// TIA Portal V19 export
FUNCTION "MANUAL INTERLOCK" : Void   // FC8, LAD
{ S7_Optimized_Access := 'TRUE' }
// stored: SetENOAutomatically false
BEGIN

REGION Network 1: ERROR BIT
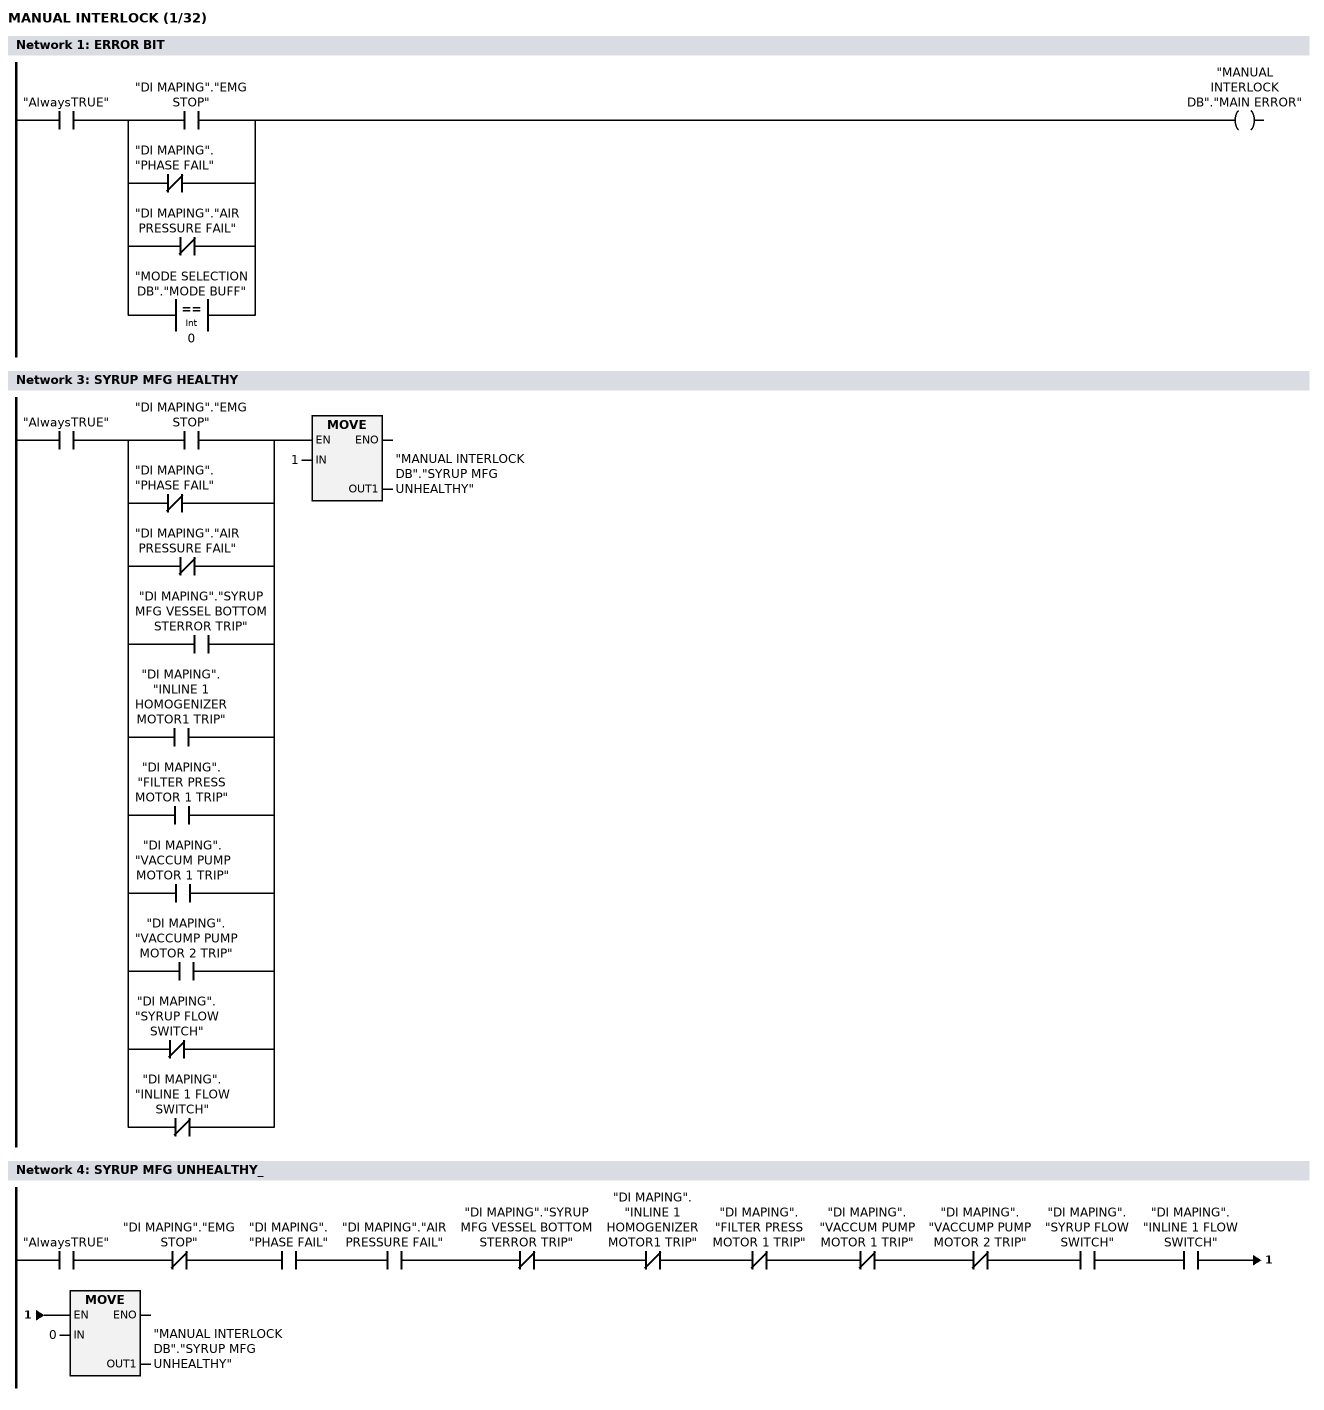
   RUNG wire#powerrail
      Contact( "AlwaysTRUE" )
      wire#w1
      Contact( "DI MAPING"."EMG STOP" )
      wire#w2
      Coil( "MANUAL INTERLOCK DB"."MAIN ERROR" )
   END_RUNG
   RUNG wire#w1
      I_Contact( "DI MAPING"."PHASE FAIL" )
   END_RUNG wire#w2
   RUNG wire#w1
      I_Contact( "DI MAPING"."AIR PRESSURE FAIL" )
   END_RUNG wire#w2
   RUNG wire#w1
      { S7_Templates := "SrcType := Int" } EQ_Contact(in1 := "MODE SELECTION DB"."MODE BUFF", in2 := 0)
   END_RUNG wire#w2
   // the same network as SCL:
   "MANUAL INTERLOCK DB"."MAIN ERROR" := "AlwaysTRUE" AND ("DI MAPING"."EMG STOP" OR NOT "DI MAPING"."PHASE FAIL" OR NOT "DI MAPING"."AIR PRESSURE FAIL" OR ("MODE SELECTION DB"."MODE BUFF" = 0));
END_REGION

REGION Network 3: SYRUP MFG HEALTHY
   RUNG wire#powerrail
      Contact( "AlwaysTRUE" )
      wire#w1
      Contact( "DI MAPING"."EMG STOP" )
      wire#w2
      Move(in := 1, out1 => "MANUAL INTERLOCK DB"."SYRUP MFG UNHEALTHY")
   END_RUNG
   RUNG wire#w1
      I_Contact( "DI MAPING"."PHASE FAIL" )
   END_RUNG wire#w2
   RUNG wire#w1
      I_Contact( "DI MAPING"."AIR PRESSURE FAIL" )
   END_RUNG wire#w2
   RUNG wire#w1
      Contact( "DI MAPING"."SYRUP MFG VESSEL BOTTOM STERROR TRIP" )
   END_RUNG wire#w2
   RUNG wire#w1
      Contact( "DI MAPING"."INLINE 1 HOMOGENIZER MOTOR1 TRIP" )
   END_RUNG wire#w2
   RUNG wire#w1
      Contact( "DI MAPING"."FILTER PRESS MOTOR 1 TRIP" )
   END_RUNG wire#w2
   RUNG wire#w1
      Contact( "DI MAPING"."VACCUM PUMP MOTOR 1 TRIP" )
   END_RUNG wire#w2
   RUNG wire#w1
      Contact( "DI MAPING"."VACCUMP PUMP MOTOR 2 TRIP" )
   END_RUNG wire#w2
   RUNG wire#w1
      I_Contact( "DI MAPING"."SYRUP FLOW SWITCH" )
   END_RUNG wire#w2
   RUNG wire#w1
      I_Contact( "DI MAPING"."INLINE 1 FLOW SWITCH" )
   END_RUNG wire#w2
   // the same network as SCL:
   IF "AlwaysTRUE" AND ("DI MAPING"."EMG STOP" OR NOT "DI MAPING"."PHASE FAIL" OR NOT "DI MAPING"."AIR PRESSURE FAIL" OR "DI MAPING"."SYRUP MFG VESSEL BOTTOM STERROR TRIP" OR "DI MAPING"."INLINE 1 HOMOGENIZER MOTOR1 TRIP" OR "DI MAPING"."FILTER PRESS MOTOR 1 TRIP" OR "DI MAPING"."VACCUM PUMP MOTOR 1 TRIP" OR "DI MAPING"."VACCUMP PUMP MOTOR 2 TRIP" OR NOT "DI MAPING"."SYRUP FLOW SWITCH" OR NOT "DI MAPING"."INLINE 1 FLOW SWITCH") THEN
       "MANUAL INTERLOCK DB"."SYRUP MFG UNHEALTHY" := 1;
   END_IF;
END_REGION

REGION Network 4: SYRUP MFG UNHEALTHY_
   RUNG wire#powerrail
      Contact( "AlwaysTRUE" )
      I_Contact( "DI MAPING"."EMG STOP" )
      Contact( "DI MAPING"."PHASE FAIL" )
      Contact( "DI MAPING"."AIR PRESSURE FAIL" )
      I_Contact( "DI MAPING"."SYRUP MFG VESSEL BOTTOM STERROR TRIP" )
      I_Contact( "DI MAPING"."INLINE 1 HOMOGENIZER MOTOR1 TRIP" )
      I_Contact( "DI MAPING"."FILTER PRESS MOTOR 1 TRIP" )
      I_Contact( "DI MAPING"."VACCUM PUMP MOTOR 1 TRIP" )
      I_Contact( "DI MAPING"."VACCUMP PUMP MOTOR 2 TRIP" )
      Contact( "DI MAPING"."SYRUP FLOW SWITCH" )
      Contact( "DI MAPING"."INLINE 1 FLOW SWITCH" )
      Move(in := 0, out1 => "MANUAL INTERLOCK DB"."SYRUP MFG UNHEALTHY")
   END_RUNG
   // the same network as SCL:
   IF "AlwaysTRUE" AND NOT "DI MAPING"."EMG STOP" AND "DI MAPING"."PHASE FAIL" AND "DI MAPING"."AIR PRESSURE FAIL" AND NOT "DI MAPING"."SYRUP MFG VESSEL BOTTOM STERROR TRIP" AND NOT "DI MAPING"."INLINE 1 HOMOGENIZER MOTOR1 TRIP" AND NOT "DI MAPING"."FILTER PRESS MOTOR 1 TRIP" AND NOT "DI MAPING"."VACCUM PUMP MOTOR 1 TRIP" AND NOT "DI MAPING"."VACCUMP PUMP MOTOR 2 TRIP" AND "DI MAPING"."SYRUP FLOW SWITCH" AND "DI MAPING"."INLINE 1 FLOW SWITCH" THEN
       "MANUAL INTERLOCK DB"."SYRUP MFG UNHEALTHY" := 0;
   END_IF;
END_REGION

REGION Network 5: PREMIXING HEALTHY
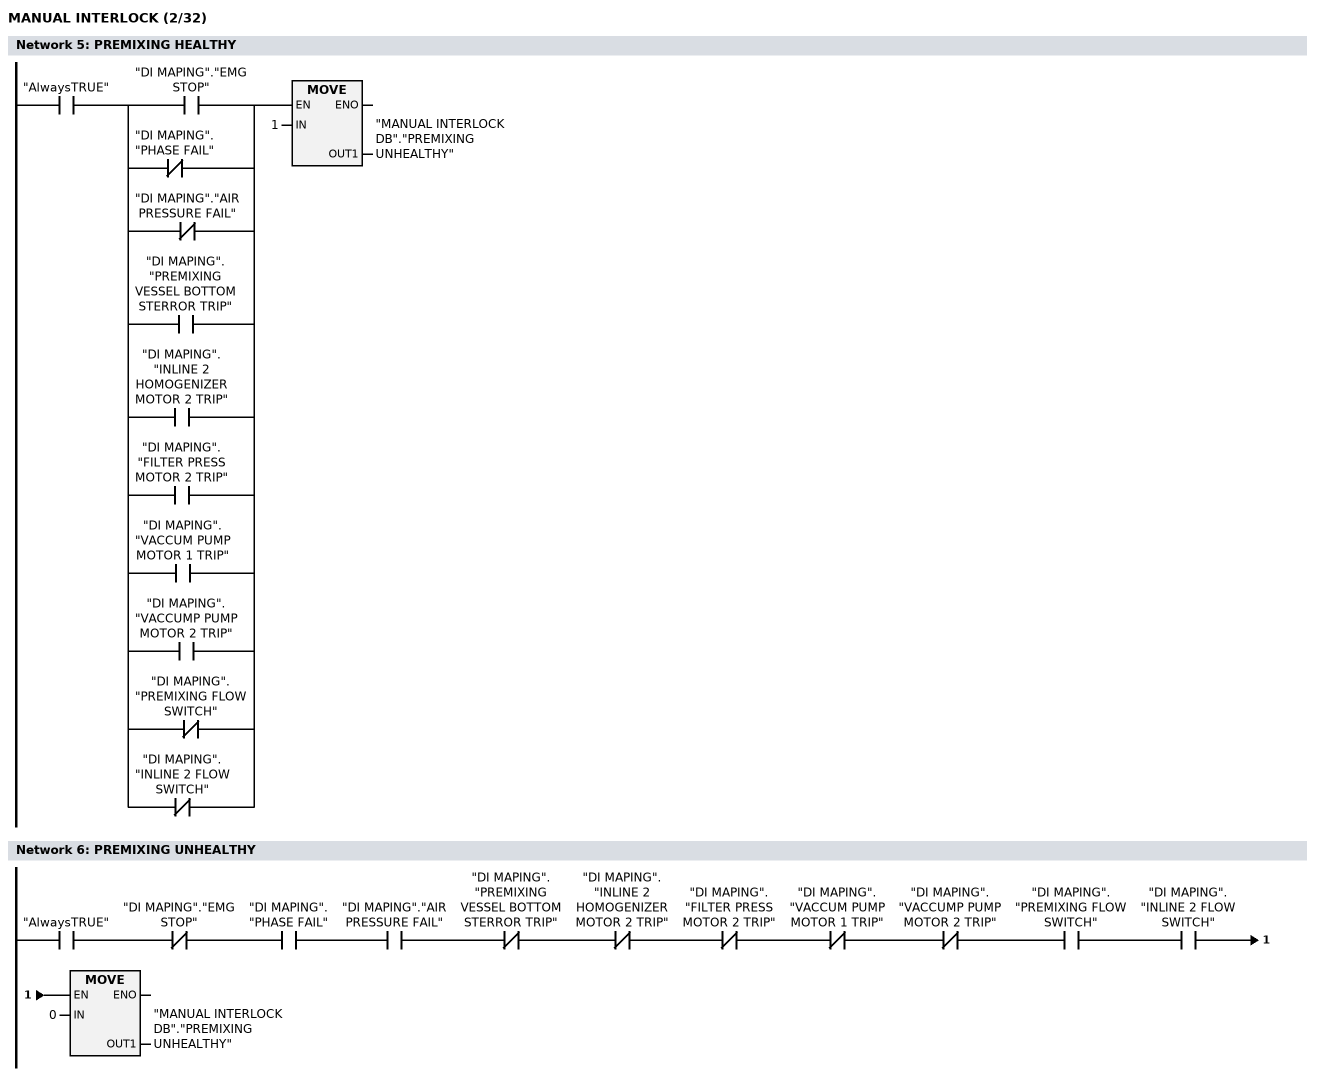
   RUNG wire#powerrail
      Contact( "AlwaysTRUE" )
      wire#w1
      Contact( "DI MAPING"."EMG STOP" )
      wire#w2
      Move(in := 1, out1 => "MANUAL INTERLOCK DB"."PREMIXING UNHEALTHY")
   END_RUNG
   RUNG wire#w1
      I_Contact( "DI MAPING"."PHASE FAIL" )
   END_RUNG wire#w2
   RUNG wire#w1
      I_Contact( "DI MAPING"."AIR PRESSURE FAIL" )
   END_RUNG wire#w2
   RUNG wire#w1
      Contact( "DI MAPING"."PREMIXING VESSEL BOTTOM STERROR TRIP" )
   END_RUNG wire#w2
   RUNG wire#w1
      Contact( "DI MAPING"."INLINE 2 HOMOGENIZER MOTOR 2 TRIP" )
   END_RUNG wire#w2
   RUNG wire#w1
      Contact( "DI MAPING"."FILTER PRESS MOTOR 2 TRIP" )
   END_RUNG wire#w2
   RUNG wire#w1
      Contact( "DI MAPING"."VACCUM PUMP MOTOR 1 TRIP" )
   END_RUNG wire#w2
   RUNG wire#w1
      Contact( "DI MAPING"."VACCUMP PUMP MOTOR 2 TRIP" )
   END_RUNG wire#w2
   RUNG wire#w1
      I_Contact( "DI MAPING"."PREMIXING FLOW SWITCH" )
   END_RUNG wire#w2
   RUNG wire#w1
      I_Contact( "DI MAPING"."INLINE 2 FLOW SWITCH" )
   END_RUNG wire#w2
   // the same network as SCL:
   IF "AlwaysTRUE" AND ("DI MAPING"."EMG STOP" OR NOT "DI MAPING"."PHASE FAIL" OR NOT "DI MAPING"."AIR PRESSURE FAIL" OR "DI MAPING"."PREMIXING VESSEL BOTTOM STERROR TRIP" OR "DI MAPING"."INLINE 2 HOMOGENIZER MOTOR 2 TRIP" OR "DI MAPING"."FILTER PRESS MOTOR 2 TRIP" OR "DI MAPING"."VACCUM PUMP MOTOR 1 TRIP" OR "DI MAPING"."VACCUMP PUMP MOTOR 2 TRIP" OR NOT "DI MAPING"."PREMIXING FLOW SWITCH" OR NOT "DI MAPING"."INLINE 2 FLOW SWITCH") THEN
       "MANUAL INTERLOCK DB"."PREMIXING UNHEALTHY" := 1;
   END_IF;
END_REGION

REGION Network 6: PREMIXING UNHEALTHY
   RUNG wire#powerrail
      Contact( "AlwaysTRUE" )
      I_Contact( "DI MAPING"."EMG STOP" )
      Contact( "DI MAPING"."PHASE FAIL" )
      Contact( "DI MAPING"."AIR PRESSURE FAIL" )
      I_Contact( "DI MAPING"."PREMIXING VESSEL BOTTOM STERROR TRIP" )
      I_Contact( "DI MAPING"."INLINE 2 HOMOGENIZER MOTOR 2 TRIP" )
      I_Contact( "DI MAPING"."FILTER PRESS MOTOR 2 TRIP" )
      I_Contact( "DI MAPING"."VACCUM PUMP MOTOR 1 TRIP" )
      I_Contact( "DI MAPING"."VACCUMP PUMP MOTOR 2 TRIP" )
      Contact( "DI MAPING"."PREMIXING FLOW SWITCH" )
      Contact( "DI MAPING"."INLINE 2 FLOW SWITCH" )
      Move(in := 0, out1 => "MANUAL INTERLOCK DB"."PREMIXING UNHEALTHY")
   END_RUNG
   // the same network as SCL:
   IF "AlwaysTRUE" AND NOT "DI MAPING"."EMG STOP" AND "DI MAPING"."PHASE FAIL" AND "DI MAPING"."AIR PRESSURE FAIL" AND NOT "DI MAPING"."PREMIXING VESSEL BOTTOM STERROR TRIP" AND NOT "DI MAPING"."INLINE 2 HOMOGENIZER MOTOR 2 TRIP" AND NOT "DI MAPING"."FILTER PRESS MOTOR 2 TRIP" AND NOT "DI MAPING"."VACCUM PUMP MOTOR 1 TRIP" AND NOT "DI MAPING"."VACCUMP PUMP MOTOR 2 TRIP" AND "DI MAPING"."PREMIXING FLOW SWITCH" AND "DI MAPING"."INLINE 2 FLOW SWITCH" THEN
       "MANUAL INTERLOCK DB"."PREMIXING UNHEALTHY" := 0;
   END_IF;
END_REGION

REGION Network 7: SUGAR HEALTHY
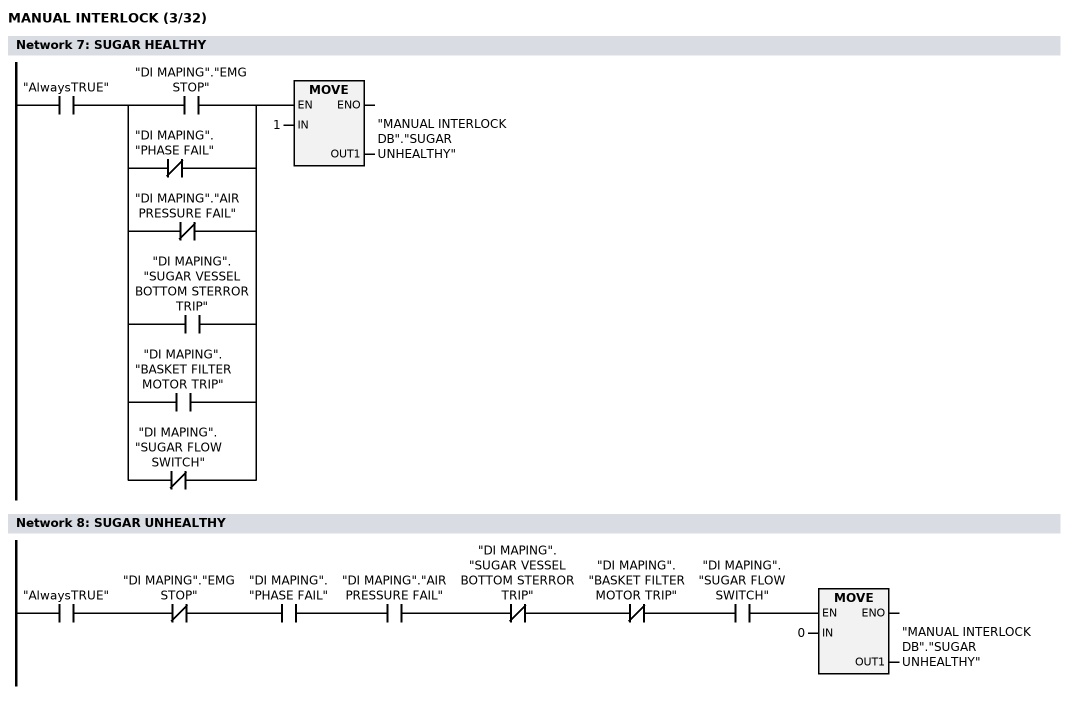
   RUNG wire#powerrail
      Contact( "AlwaysTRUE" )
      wire#w1
      Contact( "DI MAPING"."EMG STOP" )
      wire#w2
      Move(in := 1, out1 => "MANUAL INTERLOCK DB"."SUGAR UNHEALTHY")
   END_RUNG
   RUNG wire#w1
      I_Contact( "DI MAPING"."PHASE FAIL" )
   END_RUNG wire#w2
   RUNG wire#w1
      I_Contact( "DI MAPING"."AIR PRESSURE FAIL" )
   END_RUNG wire#w2
   RUNG wire#w1
      Contact( "DI MAPING"."SUGAR VESSEL BOTTOM STERROR TRIP" )
   END_RUNG wire#w2
   RUNG wire#w1
      Contact( "DI MAPING"."BASKET FILTER MOTOR TRIP" )
   END_RUNG wire#w2
   RUNG wire#w1
      I_Contact( "DI MAPING"."SUGAR FLOW SWITCH" )
   END_RUNG wire#w2
   // the same network as SCL:
   IF "AlwaysTRUE" AND ("DI MAPING"."EMG STOP" OR NOT "DI MAPING"."PHASE FAIL" OR NOT "DI MAPING"."AIR PRESSURE FAIL" OR "DI MAPING"."SUGAR VESSEL BOTTOM STERROR TRIP" OR "DI MAPING"."BASKET FILTER MOTOR TRIP" OR NOT "DI MAPING"."SUGAR FLOW SWITCH") THEN
       "MANUAL INTERLOCK DB"."SUGAR UNHEALTHY" := 1;
   END_IF;
END_REGION

REGION Network 8: SUGAR UNHEALTHY
   RUNG wire#powerrail
      Contact( "AlwaysTRUE" )
      I_Contact( "DI MAPING"."EMG STOP" )
      Contact( "DI MAPING"."PHASE FAIL" )
      Contact( "DI MAPING"."AIR PRESSURE FAIL" )
      I_Contact( "DI MAPING"."SUGAR VESSEL BOTTOM STERROR TRIP" )
      I_Contact( "DI MAPING"."BASKET FILTER MOTOR TRIP" )
      Contact( "DI MAPING"."SUGAR FLOW SWITCH" )
      Move(in := 0, out1 => "MANUAL INTERLOCK DB"."SUGAR UNHEALTHY")
   END_RUNG
   // the same network as SCL:
   IF "AlwaysTRUE" AND NOT "DI MAPING"."EMG STOP" AND "DI MAPING"."PHASE FAIL" AND "DI MAPING"."AIR PRESSURE FAIL" AND NOT "DI MAPING"."SUGAR VESSEL BOTTOM STERROR TRIP" AND NOT "DI MAPING"."BASKET FILTER MOTOR TRIP" AND "DI MAPING"."SUGAR FLOW SWITCH" THEN
       "MANUAL INTERLOCK DB"."SUGAR UNHEALTHY" := 0;
   END_IF;
END_REGION

REGION Network 10: ------------------------------------------ CONTINUE RESET-------------------------------------
END_REGION

REGION Network 11: SYRUP MFG PROCESS ERROR FOR CONTINUE
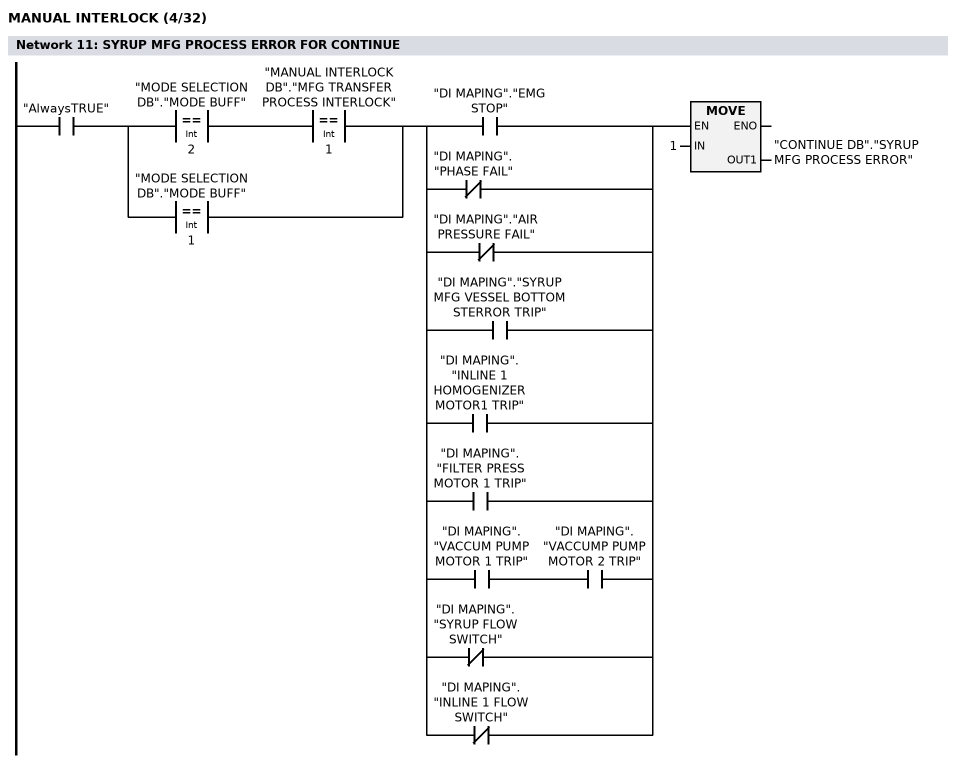
   RUNG wire#powerrail
      Contact( "AlwaysTRUE" )
      wire#w1
      { S7_Templates := "SrcType := Int" } EQ_Contact(in1 := "MODE SELECTION DB"."MODE BUFF", in2 := 2)
      { S7_Templates := "SrcType := Int" } EQ_Contact(in1 := "MANUAL INTERLOCK DB"."MFG TRANSFER PROCESS INTERLOCK", in2 := 1)
      wire#w2
      Contact( "DI MAPING"."EMG STOP" )
      wire#w3
      Move(in := 1, out1 => "CONTINUE DB"."SYRUP MFG PROCESS ERROR")
   END_RUNG
   RUNG wire#w1
      { S7_Templates := "SrcType := Int" } EQ_Contact(in1 := "MODE SELECTION DB"."MODE BUFF", in2 := 1)
   END_RUNG wire#w2
   RUNG wire#w2
      I_Contact( "DI MAPING"."PHASE FAIL" )
   END_RUNG wire#w3
   RUNG wire#w2
      I_Contact( "DI MAPING"."AIR PRESSURE FAIL" )
   END_RUNG wire#w3
   RUNG wire#w2
      Contact( "DI MAPING"."SYRUP MFG VESSEL BOTTOM STERROR TRIP" )
   END_RUNG wire#w3
   RUNG wire#w2
      Contact( "DI MAPING"."INLINE 1 HOMOGENIZER MOTOR1 TRIP" )
   END_RUNG wire#w3
   RUNG wire#w2
      Contact( "DI MAPING"."FILTER PRESS MOTOR 1 TRIP" )
   END_RUNG wire#w3
   RUNG wire#w2
      Contact( "DI MAPING"."VACCUM PUMP MOTOR 1 TRIP" )
      Contact( "DI MAPING"."VACCUMP PUMP MOTOR 2 TRIP" )
   END_RUNG wire#w3
   RUNG wire#w2
      I_Contact( "DI MAPING"."SYRUP FLOW SWITCH" )
   END_RUNG wire#w3
   RUNG wire#w2
      I_Contact( "DI MAPING"."INLINE 1 FLOW SWITCH" )
   END_RUNG wire#w3
   // the same network as SCL:
   IF "AlwaysTRUE" AND ((("MODE SELECTION DB"."MODE BUFF" = 2) AND ("MANUAL INTERLOCK DB"."MFG TRANSFER PROCESS INTERLOCK" = 1)) OR ("MODE SELECTION DB"."MODE BUFF" = 1)) AND ("DI MAPING"."EMG STOP" OR NOT "DI MAPING"."PHASE FAIL" OR NOT "DI MAPING"."AIR PRESSURE FAIL" OR "DI MAPING"."SYRUP MFG VESSEL BOTTOM STERROR TRIP" OR "DI MAPING"."INLINE 1 HOMOGENIZER MOTOR1 TRIP" OR "DI MAPING"."FILTER PRESS MOTOR 1 TRIP" OR ("DI MAPING"."VACCUM PUMP MOTOR 1 TRIP" AND "DI MAPING"."VACCUMP PUMP MOTOR 2 TRIP") OR NOT "DI MAPING"."SYRUP FLOW SWITCH" OR NOT "DI MAPING"."INLINE 1 FLOW SWITCH") THEN
       "CONTINUE DB"."SYRUP MFG PROCESS ERROR" := 1;
   END_IF;
END_REGION

REGION Network 12: PREMIXING PROCESS ERROR FOR CONTINUE
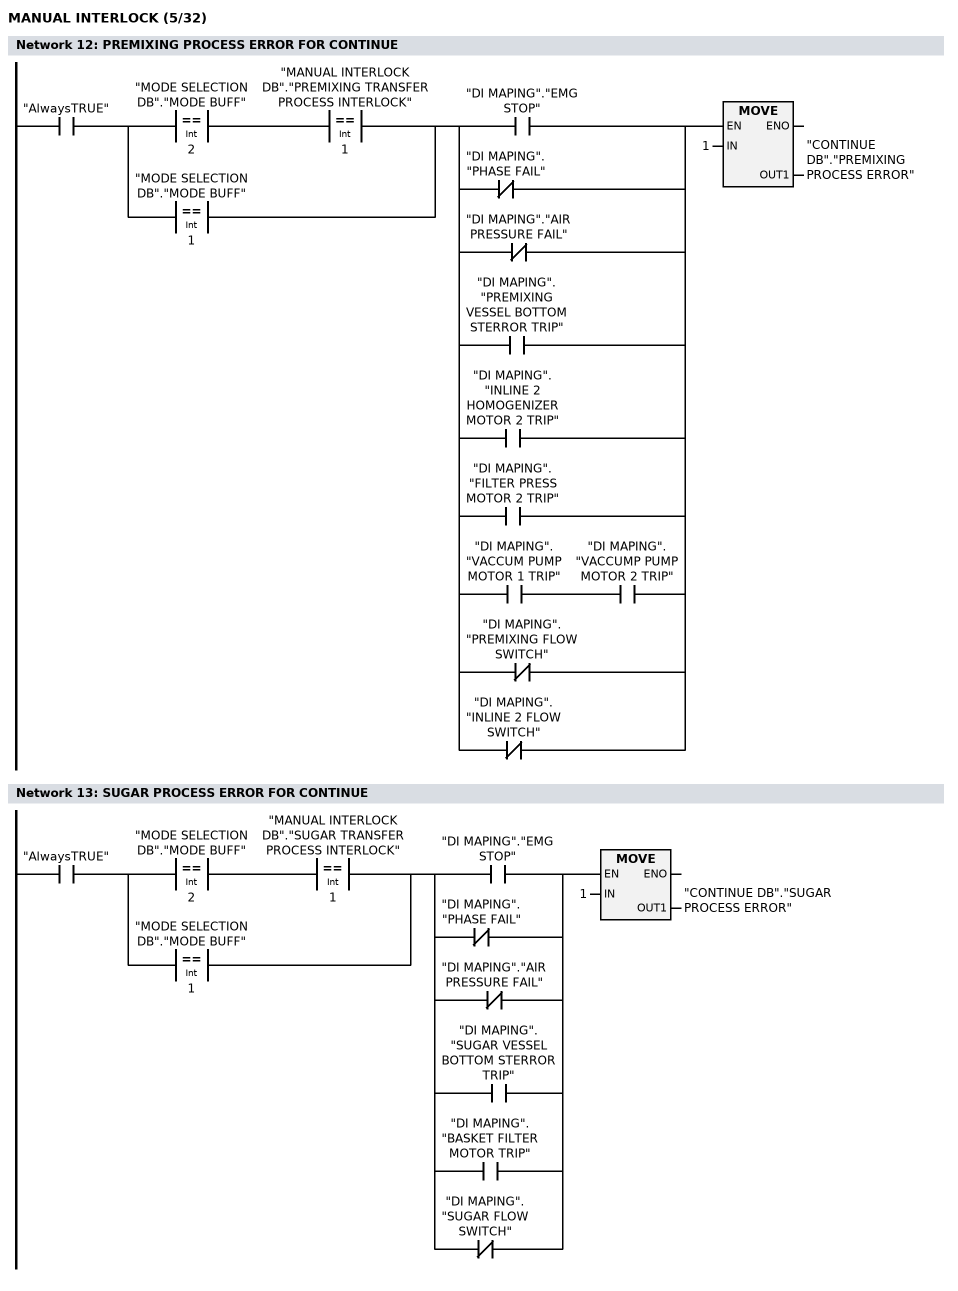
   RUNG wire#powerrail
      Contact( "AlwaysTRUE" )
      wire#w1
      { S7_Templates := "SrcType := Int" } EQ_Contact(in1 := "MODE SELECTION DB"."MODE BUFF", in2 := 2)
      { S7_Templates := "SrcType := Int" } EQ_Contact(in1 := "MANUAL INTERLOCK DB"."PREMIXING TRANSFER PROCESS INTERLOCK", in2 := 1)
      wire#w2
      Contact( "DI MAPING"."EMG STOP" )
      wire#w3
      Move(in := 1, out1 => "CONTINUE DB"."PREMIXING PROCESS ERROR")
   END_RUNG
   RUNG wire#w1
      { S7_Templates := "SrcType := Int" } EQ_Contact(in1 := "MODE SELECTION DB"."MODE BUFF", in2 := 1)
   END_RUNG wire#w2
   RUNG wire#w2
      I_Contact( "DI MAPING"."PHASE FAIL" )
   END_RUNG wire#w3
   RUNG wire#w2
      I_Contact( "DI MAPING"."AIR PRESSURE FAIL" )
   END_RUNG wire#w3
   RUNG wire#w2
      Contact( "DI MAPING"."PREMIXING VESSEL BOTTOM STERROR TRIP" )
   END_RUNG wire#w3
   RUNG wire#w2
      Contact( "DI MAPING"."INLINE 2 HOMOGENIZER MOTOR 2 TRIP" )
   END_RUNG wire#w3
   RUNG wire#w2
      Contact( "DI MAPING"."FILTER PRESS MOTOR 2 TRIP" )
   END_RUNG wire#w3
   RUNG wire#w2
      Contact( "DI MAPING"."VACCUM PUMP MOTOR 1 TRIP" )
      Contact( "DI MAPING"."VACCUMP PUMP MOTOR 2 TRIP" )
   END_RUNG wire#w3
   RUNG wire#w2
      I_Contact( "DI MAPING"."PREMIXING FLOW SWITCH" )
   END_RUNG wire#w3
   RUNG wire#w2
      I_Contact( "DI MAPING"."INLINE 2 FLOW SWITCH" )
   END_RUNG wire#w3
   // the same network as SCL:
   IF "AlwaysTRUE" AND ((("MODE SELECTION DB"."MODE BUFF" = 2) AND ("MANUAL INTERLOCK DB"."PREMIXING TRANSFER PROCESS INTERLOCK" = 1)) OR ("MODE SELECTION DB"."MODE BUFF" = 1)) AND ("DI MAPING"."EMG STOP" OR NOT "DI MAPING"."PHASE FAIL" OR NOT "DI MAPING"."AIR PRESSURE FAIL" OR "DI MAPING"."PREMIXING VESSEL BOTTOM STERROR TRIP" OR "DI MAPING"."INLINE 2 HOMOGENIZER MOTOR 2 TRIP" OR "DI MAPING"."FILTER PRESS MOTOR 2 TRIP" OR ("DI MAPING"."VACCUM PUMP MOTOR 1 TRIP" AND "DI MAPING"."VACCUMP PUMP MOTOR 2 TRIP") OR NOT "DI MAPING"."PREMIXING FLOW SWITCH" OR NOT "DI MAPING"."INLINE 2 FLOW SWITCH") THEN
       "CONTINUE DB"."PREMIXING PROCESS ERROR" := 1;
   END_IF;
END_REGION

REGION Network 13: SUGAR PROCESS ERROR FOR CONTINUE
   RUNG wire#powerrail
      Contact( "AlwaysTRUE" )
      wire#w1
      { S7_Templates := "SrcType := Int" } EQ_Contact(in1 := "MODE SELECTION DB"."MODE BUFF", in2 := 2)
      { S7_Templates := "SrcType := Int" } EQ_Contact(in1 := "MANUAL INTERLOCK DB"."SUGAR TRANSFER PROCESS INTERLOCK", in2 := 1)
      wire#w2
      Contact( "DI MAPING"."EMG STOP" )
      wire#w3
      Move(in := 1, out1 => "CONTINUE DB"."SUGAR PROCESS ERROR")
   END_RUNG
   RUNG wire#w1
      { S7_Templates := "SrcType := Int" } EQ_Contact(in1 := "MODE SELECTION DB"."MODE BUFF", in2 := 1)
   END_RUNG wire#w2
   RUNG wire#w2
      I_Contact( "DI MAPING"."PHASE FAIL" )
   END_RUNG wire#w3
   RUNG wire#w2
      I_Contact( "DI MAPING"."AIR PRESSURE FAIL" )
   END_RUNG wire#w3
   RUNG wire#w2
      Contact( "DI MAPING"."SUGAR VESSEL BOTTOM STERROR TRIP" )
   END_RUNG wire#w3
   RUNG wire#w2
      Contact( "DI MAPING"."BASKET FILTER MOTOR TRIP" )
   END_RUNG wire#w3
   RUNG wire#w2
      I_Contact( "DI MAPING"."SUGAR FLOW SWITCH" )
   END_RUNG wire#w3
   // the same network as SCL:
   IF "AlwaysTRUE" AND ((("MODE SELECTION DB"."MODE BUFF" = 2) AND ("MANUAL INTERLOCK DB"."SUGAR TRANSFER PROCESS INTERLOCK" = 1)) OR ("MODE SELECTION DB"."MODE BUFF" = 1)) AND ("DI MAPING"."EMG STOP" OR NOT "DI MAPING"."PHASE FAIL" OR NOT "DI MAPING"."AIR PRESSURE FAIL" OR "DI MAPING"."SUGAR VESSEL BOTTOM STERROR TRIP" OR "DI MAPING"."BASKET FILTER MOTOR TRIP" OR NOT "DI MAPING"."SUGAR FLOW SWITCH") THEN
       "CONTINUE DB"."SUGAR PROCESS ERROR" := 1;
   END_IF;
END_REGION

REGION Network 15: CONTINUE PROCESS-SYRUP MFG
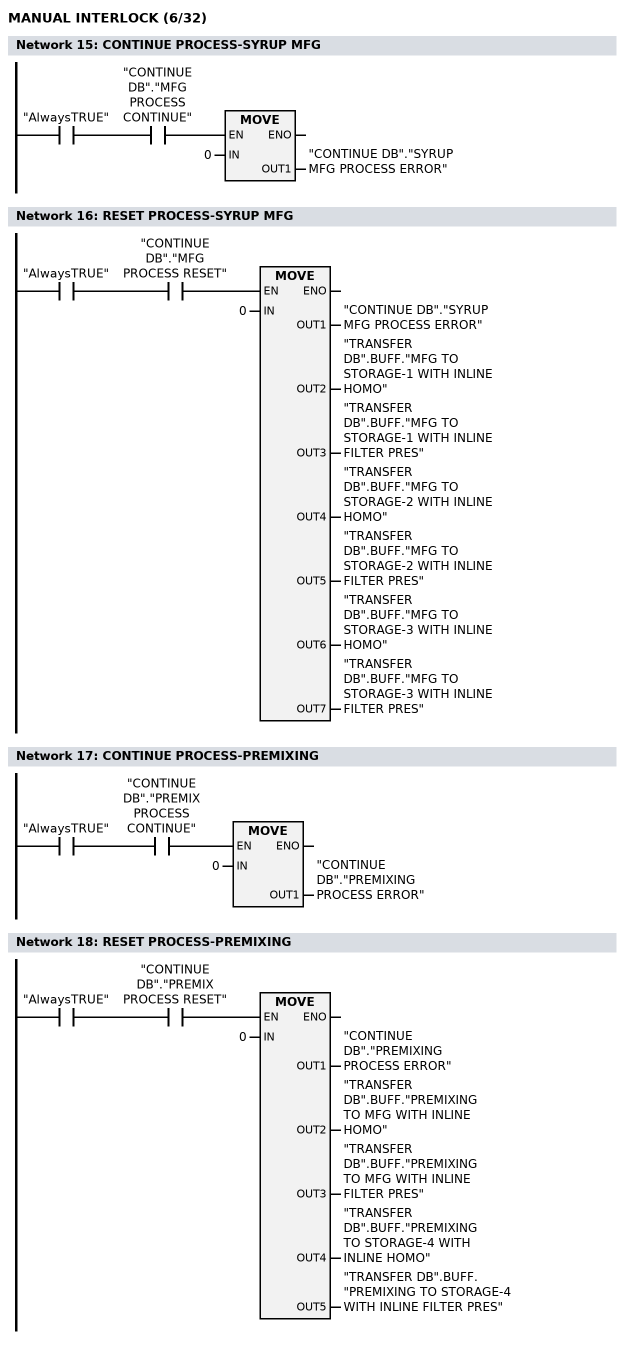
   RUNG wire#powerrail
      Contact( "AlwaysTRUE" )
      Contact( "CONTINUE DB"."MFG PROCESS CONTINUE" )
      Move(in := 0, out1 => "CONTINUE DB"."SYRUP MFG PROCESS ERROR")
   END_RUNG
   // the same network as SCL:
   IF "AlwaysTRUE" AND "CONTINUE DB"."MFG PROCESS CONTINUE" THEN
       "CONTINUE DB"."SYRUP MFG PROCESS ERROR" := 0;
   END_IF;
END_REGION

REGION Network 16: RESET PROCESS-SYRUP MFG
   RUNG wire#powerrail
      Contact( "AlwaysTRUE" )
      Contact( "CONTINUE DB"."MFG PROCESS RESET" )
      Move(in := 0, out1 => "CONTINUE DB"."SYRUP MFG PROCESS ERROR", out2 => "TRANSFER DB".BUFF."MFG TO STORAGE-1 WITH INLINE HOMO", out3 => "TRANSFER DB".BUFF."MFG TO STORAGE-1 WITH INLINE FILTER PRES", out4 => "TRANSFER DB".BUFF."MFG TO STORAGE-2 WITH INLINE HOMO", out5 => "TRANSFER DB".BUFF."MFG TO STORAGE-2 WITH INLINE FILTER PRES", out6 => "TRANSFER DB".BUFF."MFG TO STORAGE-3 WITH INLINE HOMO", out7 => "TRANSFER DB".BUFF."MFG TO STORAGE-3 WITH INLINE FILTER PRES")
   END_RUNG
   // the same network as SCL:
   IF "AlwaysTRUE" AND "CONTINUE DB"."MFG PROCESS RESET" THEN
       "CONTINUE DB"."SYRUP MFG PROCESS ERROR" := 0;
       "TRANSFER DB".BUFF."MFG TO STORAGE-1 WITH INLINE HOMO" := 0;
       "TRANSFER DB".BUFF."MFG TO STORAGE-1 WITH INLINE FILTER PRES" := 0;
       "TRANSFER DB".BUFF."MFG TO STORAGE-2 WITH INLINE HOMO" := 0;
       "TRANSFER DB".BUFF."MFG TO STORAGE-2 WITH INLINE FILTER PRES" := 0;
       "TRANSFER DB".BUFF."MFG TO STORAGE-3 WITH INLINE HOMO" := 0;
       "TRANSFER DB".BUFF."MFG TO STORAGE-3 WITH INLINE FILTER PRES" := 0;
   END_IF;
END_REGION

REGION Network 17: CONTINUE PROCESS-PREMIXING
   RUNG wire#powerrail
      Contact( "AlwaysTRUE" )
      Contact( "CONTINUE DB"."PREMIX PROCESS CONTINUE" )
      Move(in := 0, out1 => "CONTINUE DB"."PREMIXING PROCESS ERROR")
   END_RUNG
   // the same network as SCL:
   IF "AlwaysTRUE" AND "CONTINUE DB"."PREMIX PROCESS CONTINUE" THEN
       "CONTINUE DB"."PREMIXING PROCESS ERROR" := 0;
   END_IF;
END_REGION

REGION Network 18: RESET PROCESS-PREMIXING
   RUNG wire#powerrail
      Contact( "AlwaysTRUE" )
      Contact( "CONTINUE DB"."PREMIX PROCESS RESET" )
      Move(in := 0, out1 => "CONTINUE DB"."PREMIXING PROCESS ERROR", out2 => "TRANSFER DB".BUFF."PREMIXING TO MFG WITH INLINE HOMO", out3 => "TRANSFER DB".BUFF."PREMIXING TO MFG WITH INLINE FILTER PRES", out4 => "TRANSFER DB".BUFF."PREMIXING TO STORAGE-4 WITH INLINE HOMO", out5 => "TRANSFER DB".BUFF."PREMIXING TO STORAGE-4 WITH INLINE FILTER PRES")
   END_RUNG
   // the same network as SCL:
   IF "AlwaysTRUE" AND "CONTINUE DB"."PREMIX PROCESS RESET" THEN
       "CONTINUE DB"."PREMIXING PROCESS ERROR" := 0;
       "TRANSFER DB".BUFF."PREMIXING TO MFG WITH INLINE HOMO" := 0;
       "TRANSFER DB".BUFF."PREMIXING TO MFG WITH INLINE FILTER PRES" := 0;
       "TRANSFER DB".BUFF."PREMIXING TO STORAGE-4 WITH INLINE HOMO" := 0;
       "TRANSFER DB".BUFF."PREMIXING TO STORAGE-4 WITH INLINE FILTER PRES" := 0;
   END_IF;
END_REGION

REGION Network 19: CONTINUE PROCESS-SUGAR
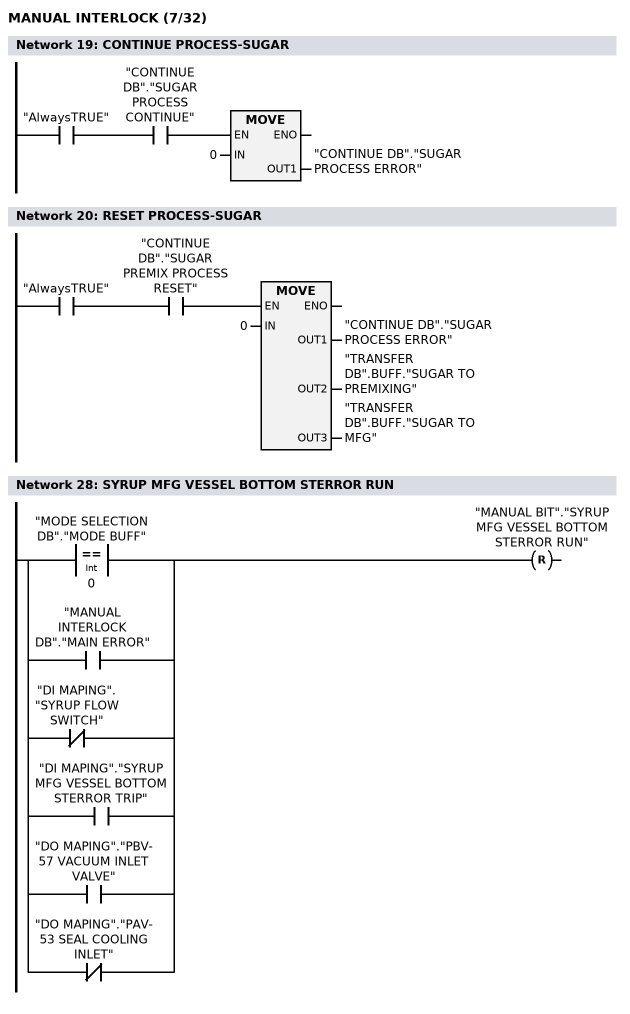
   RUNG wire#powerrail
      Contact( "AlwaysTRUE" )
      Contact( "CONTINUE DB"."SUGAR PROCESS CONTINUE" )
      Move(in := 0, out1 => "CONTINUE DB"."SUGAR PROCESS ERROR")
   END_RUNG
   // the same network as SCL:
   IF "AlwaysTRUE" AND "CONTINUE DB"."SUGAR PROCESS CONTINUE" THEN
       "CONTINUE DB"."SUGAR PROCESS ERROR" := 0;
   END_IF;
END_REGION

REGION Network 20: RESET PROCESS-SUGAR
   RUNG wire#powerrail
      Contact( "AlwaysTRUE" )
      Contact( "CONTINUE DB"."SUGAR PREMIX PROCESS RESET" )
      Move(in := 0, out1 => "CONTINUE DB"."SUGAR PROCESS ERROR", out2 => "TRANSFER DB".BUFF."SUGAR TO PREMIXING", out3 => "TRANSFER DB".BUFF."SUGAR TO MFG")
   END_RUNG
   // the same network as SCL:
   IF "AlwaysTRUE" AND "CONTINUE DB"."SUGAR PREMIX PROCESS RESET" THEN
       "CONTINUE DB"."SUGAR PROCESS ERROR" := 0;
       "TRANSFER DB".BUFF."SUGAR TO PREMIXING" := 0;
       "TRANSFER DB".BUFF."SUGAR TO MFG" := 0;
   END_IF;
END_REGION

REGION Network 22: ------------------------------TRANSFER PROCESS INTERLOCK---------------------------------------
END_REGION

REGION Network 23 (SCL): MFG TRANSFER PROCESS INTERLOCK
   IF 
       "TRANSFER DB".BUFF."MFG TO STORAGE-1 WITH INLINE HOMO" <> 0 OR
       "TRANSFER DB".BUFF."MFG TO STORAGE-1 WITH INLINE FILTER PRES" <> 0 OR
       "TRANSFER DB".BUFF."MFG TO STORAGE-2 WITH INLINE HOMO" <> 0 OR
       "TRANSFER DB".BUFF."MFG TO STORAGE-2 WITH INLINE FILTER PRES" <> 0 OR
       "TRANSFER DB".BUFF."MFG TO STORAGE-3 WITH INLINE HOMO" <> 0 OR
       "TRANSFER DB".BUFF."MFG TO STORAGE-3 WITH INLINE FILTER PRES" <> 0
   THEN
       "MANUAL INTERLOCK DB"."MFG TRANSFER PROCESS INTERLOCK" := 1;
   ELSIF "TRANSFER DB"."MFG VACCUM PUMP MOTOR-W 1 BIT"<>0
       OR "TRANSFER DB"."MFG VACCUMP PUMP MOTOR-S2 BIT"<>0
   THEN
       "MANUAL INTERLOCK DB"."MFG TRANSFER PROCESS INTERLOCK" := 2;
   ELSIF "RECIRCULATION DB".MFG.BUFF<>0
   THEN
       "MANUAL INTERLOCK DB"."MFG TRANSFER PROCESS INTERLOCK" := 3;
   ELSE
       "MANUAL INTERLOCK DB"."MFG TRANSFER PROCESS INTERLOCK" := 0;
   END_IF;
END_REGION

REGION Network 24 (SCL): PREMIXING TRANSFER PROCESS INTERLOCK
   IF
       "TRANSFER DB".BUFF."PREMIXING TO MFG WITH INLINE HOMO" <> 0 OR
       "TRANSFER DB".BUFF."PREMIXING TO MFG WITH INLINE FILTER PRES" <> 0 OR
       "TRANSFER DB".BUFF."PREMIXING TO STORAGE-4 WITH INLINE HOMO" <> 0 OR
       "TRANSFER DB".BUFF."PREMIXING TO STORAGE-4 WITH INLINE FILTER PRES" <> 0
   THEN
       "MANUAL INTERLOCK DB"."PREMIXING TRANSFER PROCESS INTERLOCK" := 1;
   ELSIF "TRANSFER DB"."PREMIXING VACCUM PUMP MOTOR-W 1 BIT"<>0 OR
       "TRANSFER DB"."PREMIXING VACCUMP PUMP MOTOR-S2 BIT"
   THEN
       "MANUAL INTERLOCK DB"."PREMIXING TRANSFER PROCESS INTERLOCK" := 2;
   ELSIF "RECIRCULATION DB".PREMIXING.BUFF<>0
   THEN
       "MANUAL INTERLOCK DB"."PREMIXING TRANSFER PROCESS INTERLOCK" := 3;
   ELSE
       "MANUAL INTERLOCK DB"."PREMIXING TRANSFER PROCESS INTERLOCK" := 0;
   END_IF;
END_REGION

REGION Network 25 (SCL): SUGAR TRANSFER PROCESS INTERLOCK
   IF "TRANSFER DB".BUFF."SUGAR TO PREMIXING" <>0 OR
       "TRANSFER DB".BUFF."SUGAR TO MFG"<>0
   THEN
       "MANUAL INTERLOCK DB"."SUGAR TRANSFER PROCESS INTERLOCK" := 1;
   ELSIF "DO MAPING"."PBV-30 VACUUM INLET VALVE" <>0
   THEN
       "MANUAL INTERLOCK DB"."SUGAR TRANSFER PROCESS INTERLOCK" := 2;
   ELSE
       "MANUAL INTERLOCK DB"."SUGAR TRANSFER PROCESS INTERLOCK" := 0;

   END_IF;
END_REGION

REGION Network 27: ------------------------------------------ MANUAL BIT RESET-------------------------------------
END_REGION

REGION Network 28: SYRUP MFG VESSEL BOTTOM STERROR RUN
   RUNG wire#powerrail
      { S7_Templates := "SrcType := Int" } EQ_Contact(in1 := "MODE SELECTION DB"."MODE BUFF", in2 := 0)
      wire#w1
      R_Coil( "MANUAL BIT"."SYRUP MFG VESSEL BOTTOM STERROR RUN" )
   END_RUNG
   RUNG wire#powerrail
      Contact( "MANUAL INTERLOCK DB"."MAIN ERROR" )
   END_RUNG wire#w1
   RUNG wire#powerrail
      I_Contact( "DI MAPING"."SYRUP FLOW SWITCH" )
   END_RUNG wire#w1
   RUNG wire#powerrail
      Contact( "DI MAPING"."SYRUP MFG VESSEL BOTTOM STERROR TRIP" )
   END_RUNG wire#w1
   RUNG wire#powerrail
      Contact( "DO MAPING"."PBV-57 VACUUM INLET VALVE" )
   END_RUNG wire#w1
   RUNG wire#powerrail
      I_Contact( "DO MAPING"."PAV-53 SEAL COOLING INLET" )
   END_RUNG wire#w1
   // the same network as SCL:
   IF ("MODE SELECTION DB"."MODE BUFF" = 0) OR "MANUAL INTERLOCK DB"."MAIN ERROR" OR NOT "DI MAPING"."SYRUP FLOW SWITCH" OR "DI MAPING"."SYRUP MFG VESSEL BOTTOM STERROR TRIP" OR "DO MAPING"."PBV-57 VACUUM INLET VALVE" OR NOT "DO MAPING"."PAV-53 SEAL COOLING INLET" THEN
       "MANUAL BIT"."SYRUP MFG VESSEL BOTTOM STERROR RUN" := FALSE;
   END_IF;
END_REGION

REGION Network 29: PREMIXING VESSEL BOTTOM STERROR RUN
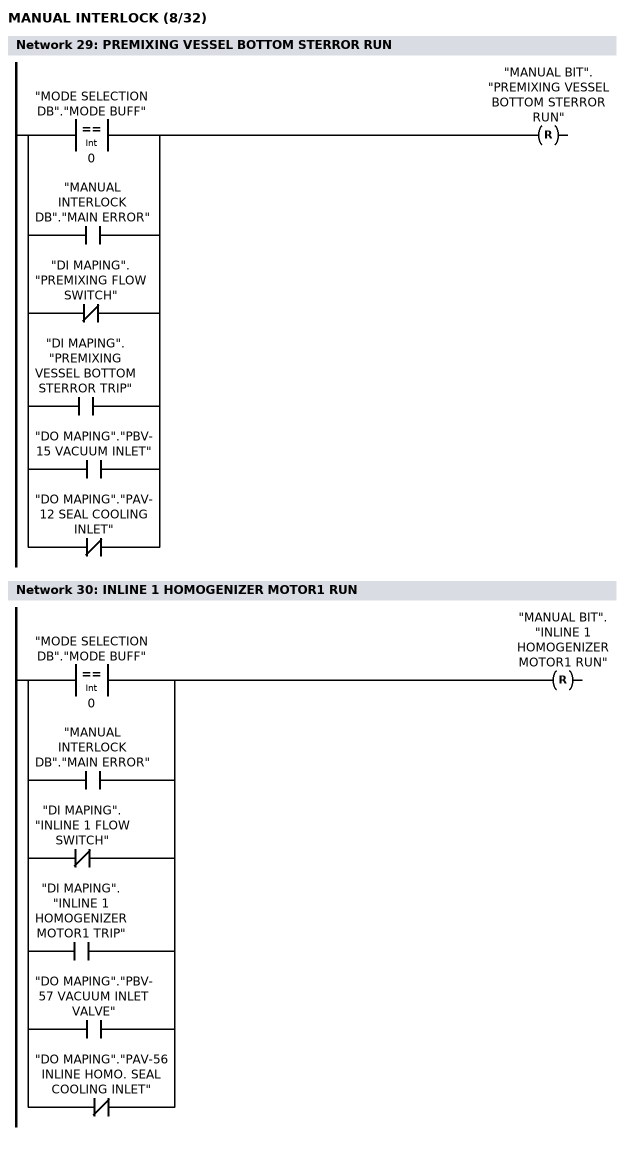
   RUNG wire#powerrail
      { S7_Templates := "SrcType := Int" } EQ_Contact(in1 := "MODE SELECTION DB"."MODE BUFF", in2 := 0)
      wire#w1
      R_Coil( "MANUAL BIT"."PREMIXING VESSEL BOTTOM STERROR RUN" )
   END_RUNG
   RUNG wire#powerrail
      Contact( "MANUAL INTERLOCK DB"."MAIN ERROR" )
   END_RUNG wire#w1
   RUNG wire#powerrail
      I_Contact( "DI MAPING"."PREMIXING FLOW SWITCH" )
   END_RUNG wire#w1
   RUNG wire#powerrail
      Contact( "DI MAPING"."PREMIXING VESSEL BOTTOM STERROR TRIP" )
   END_RUNG wire#w1
   RUNG wire#powerrail
      Contact( "DO MAPING"."PBV-15 VACUUM INLET" )
   END_RUNG wire#w1
   RUNG wire#powerrail
      I_Contact( "DO MAPING"."PAV-12 SEAL COOLING INLET" )
   END_RUNG wire#w1
   // the same network as SCL:
   IF ("MODE SELECTION DB"."MODE BUFF" = 0) OR "MANUAL INTERLOCK DB"."MAIN ERROR" OR NOT "DI MAPING"."PREMIXING FLOW SWITCH" OR "DI MAPING"."PREMIXING VESSEL BOTTOM STERROR TRIP" OR "DO MAPING"."PBV-15 VACUUM INLET" OR NOT "DO MAPING"."PAV-12 SEAL COOLING INLET" THEN
       "MANUAL BIT"."PREMIXING VESSEL BOTTOM STERROR RUN" := FALSE;
   END_IF;
END_REGION

REGION Network 30: INLINE 1 HOMOGENIZER MOTOR1 RUN
   RUNG wire#powerrail
      { S7_Templates := "SrcType := Int" } EQ_Contact(in1 := "MODE SELECTION DB"."MODE BUFF", in2 := 0)
      wire#w1
      R_Coil( "MANUAL BIT"."INLINE 1 HOMOGENIZER MOTOR1 RUN" )
   END_RUNG
   RUNG wire#powerrail
      Contact( "MANUAL INTERLOCK DB"."MAIN ERROR" )
   END_RUNG wire#w1
   RUNG wire#powerrail
      I_Contact( "DI MAPING"."INLINE 1 FLOW SWITCH" )
   END_RUNG wire#w1
   RUNG wire#powerrail
      Contact( "DI MAPING"."INLINE 1 HOMOGENIZER MOTOR1 TRIP" )
   END_RUNG wire#w1
   RUNG wire#powerrail
      Contact( "DO MAPING"."PBV-57 VACUUM INLET VALVE" )
   END_RUNG wire#w1
   RUNG wire#powerrail
      I_Contact( "DO MAPING"."PAV-56 INLINE HOMO. SEAL COOLING INLET" )
   END_RUNG wire#w1
   // the same network as SCL:
   IF ("MODE SELECTION DB"."MODE BUFF" = 0) OR "MANUAL INTERLOCK DB"."MAIN ERROR" OR NOT "DI MAPING"."INLINE 1 FLOW SWITCH" OR "DI MAPING"."INLINE 1 HOMOGENIZER MOTOR1 TRIP" OR "DO MAPING"."PBV-57 VACUUM INLET VALVE" OR NOT "DO MAPING"."PAV-56 INLINE HOMO. SEAL COOLING INLET" THEN
       "MANUAL BIT"."INLINE 1 HOMOGENIZER MOTOR1 RUN" := FALSE;
   END_IF;
END_REGION

REGION Network 31: INLINE 2 HOMOGENIZER MOTOR 2 RUN
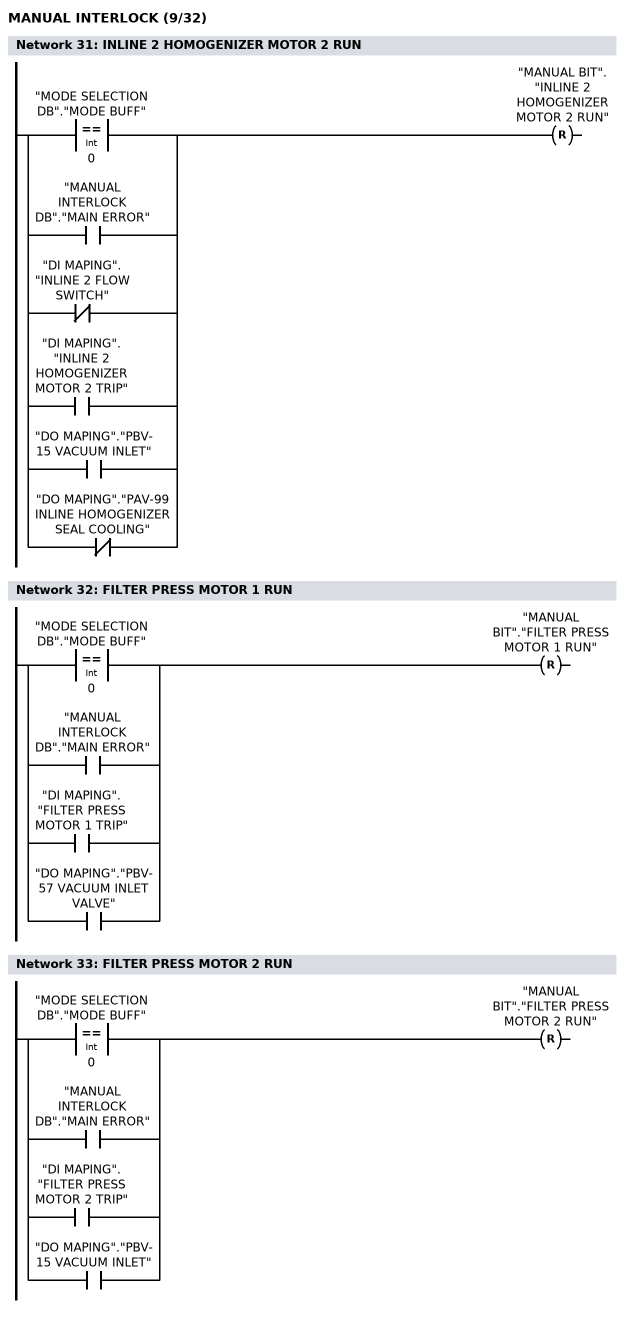
   RUNG wire#powerrail
      { S7_Templates := "SrcType := Int" } EQ_Contact(in1 := "MODE SELECTION DB"."MODE BUFF", in2 := 0)
      wire#w1
      R_Coil( "MANUAL BIT"."INLINE 2 HOMOGENIZER MOTOR 2 RUN" )
   END_RUNG
   RUNG wire#powerrail
      Contact( "MANUAL INTERLOCK DB"."MAIN ERROR" )
   END_RUNG wire#w1
   RUNG wire#powerrail
      I_Contact( "DI MAPING"."INLINE 2 FLOW SWITCH" )
   END_RUNG wire#w1
   RUNG wire#powerrail
      Contact( "DI MAPING"."INLINE 2 HOMOGENIZER MOTOR 2 TRIP" )
   END_RUNG wire#w1
   RUNG wire#powerrail
      Contact( "DO MAPING"."PBV-15 VACUUM INLET" )
   END_RUNG wire#w1
   RUNG wire#powerrail
      I_Contact( "DO MAPING"."PAV-99 INLINE HOMOGENIZER SEAL COOLING" )
   END_RUNG wire#w1
   // the same network as SCL:
   IF ("MODE SELECTION DB"."MODE BUFF" = 0) OR "MANUAL INTERLOCK DB"."MAIN ERROR" OR NOT "DI MAPING"."INLINE 2 FLOW SWITCH" OR "DI MAPING"."INLINE 2 HOMOGENIZER MOTOR 2 TRIP" OR "DO MAPING"."PBV-15 VACUUM INLET" OR NOT "DO MAPING"."PAV-99 INLINE HOMOGENIZER SEAL COOLING" THEN
       "MANUAL BIT"."INLINE 2 HOMOGENIZER MOTOR 2 RUN" := FALSE;
   END_IF;
END_REGION

REGION Network 32: FILTER PRESS MOTOR 1 RUN
   RUNG wire#powerrail
      { S7_Templates := "SrcType := Int" } EQ_Contact(in1 := "MODE SELECTION DB"."MODE BUFF", in2 := 0)
      wire#w1
      R_Coil( "MANUAL BIT"."FILTER PRESS MOTOR 1 RUN" )
   END_RUNG
   RUNG wire#powerrail
      Contact( "MANUAL INTERLOCK DB"."MAIN ERROR" )
   END_RUNG wire#w1
   RUNG wire#powerrail
      Contact( "DI MAPING"."FILTER PRESS MOTOR 1 TRIP" )
   END_RUNG wire#w1
   RUNG wire#powerrail
      Contact( "DO MAPING"."PBV-57 VACUUM INLET VALVE" )
   END_RUNG wire#w1
   // the same network as SCL:
   IF ("MODE SELECTION DB"."MODE BUFF" = 0) OR "MANUAL INTERLOCK DB"."MAIN ERROR" OR "DI MAPING"."FILTER PRESS MOTOR 1 TRIP" OR "DO MAPING"."PBV-57 VACUUM INLET VALVE" THEN
       "MANUAL BIT"."FILTER PRESS MOTOR 1 RUN" := FALSE;
   END_IF;
END_REGION

REGION Network 33: FILTER PRESS MOTOR 2 RUN
   RUNG wire#powerrail
      { S7_Templates := "SrcType := Int" } EQ_Contact(in1 := "MODE SELECTION DB"."MODE BUFF", in2 := 0)
      wire#w1
      R_Coil( "MANUAL BIT"."FILTER PRESS MOTOR 2 RUN" )
   END_RUNG
   RUNG wire#powerrail
      Contact( "MANUAL INTERLOCK DB"."MAIN ERROR" )
   END_RUNG wire#w1
   RUNG wire#powerrail
      Contact( "DI MAPING"."FILTER PRESS MOTOR 2 TRIP" )
   END_RUNG wire#w1
   RUNG wire#powerrail
      Contact( "DO MAPING"."PBV-15 VACUUM INLET" )
   END_RUNG wire#w1
   // the same network as SCL:
   IF ("MODE SELECTION DB"."MODE BUFF" = 0) OR "MANUAL INTERLOCK DB"."MAIN ERROR" OR "DI MAPING"."FILTER PRESS MOTOR 2 TRIP" OR "DO MAPING"."PBV-15 VACUUM INLET" THEN
       "MANUAL BIT"."FILTER PRESS MOTOR 2 RUN" := FALSE;
   END_IF;
END_REGION

REGION Network 34: VACCUM PUMP MOTOR 1 RUN
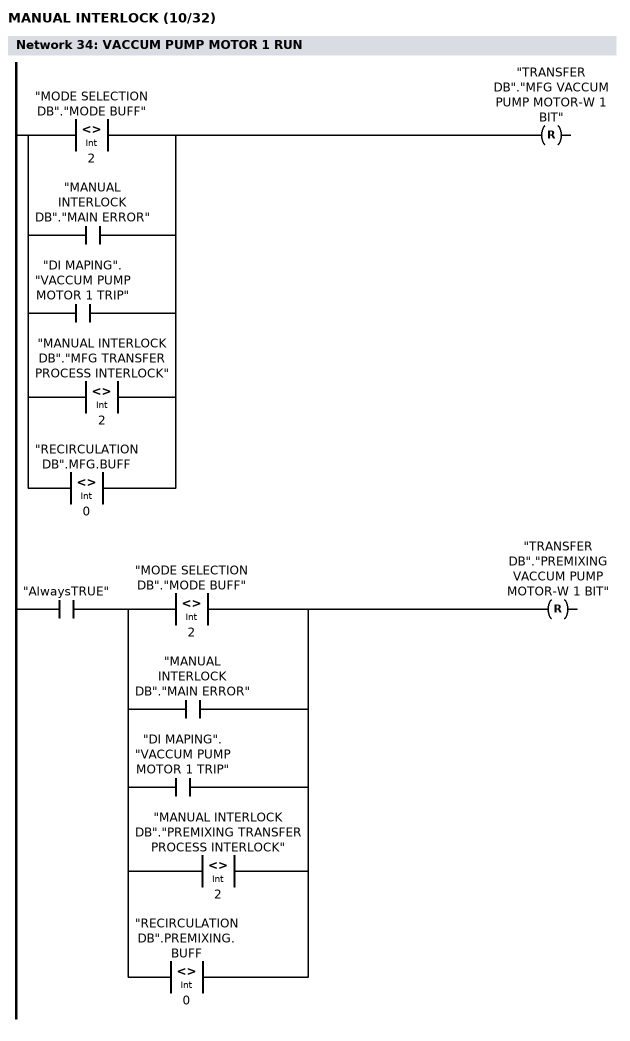
   RUNG wire#powerrail
      { S7_Templates := "SrcType := Int" } NE_Contact(in1 := "MODE SELECTION DB"."MODE BUFF", in2 := 2)
      wire#w1
      R_Coil( "TRANSFER DB"."MFG VACCUM PUMP MOTOR-W 1 BIT" )
   END_RUNG
   RUNG wire#powerrail
      Contact( "MANUAL INTERLOCK DB"."MAIN ERROR" )
   END_RUNG wire#w1
   RUNG wire#powerrail
      Contact( "DI MAPING"."VACCUM PUMP MOTOR 1 TRIP" )
   END_RUNG wire#w1
   RUNG wire#powerrail
      { S7_Templates := "SrcType := Int" } NE_Contact(in1 := "MANUAL INTERLOCK DB"."MFG TRANSFER PROCESS INTERLOCK", in2 := 2)
   END_RUNG wire#w1
   RUNG wire#powerrail
      { S7_Templates := "SrcType := Int" } NE_Contact(in1 := "RECIRCULATION DB".MFG.BUFF, in2 := 0)
   END_RUNG wire#w1
   RUNG wire#powerrail
      Contact( "AlwaysTRUE" )
      wire#w2
      { S7_Templates := "SrcType := Int" } NE_Contact(in1 := "MODE SELECTION DB"."MODE BUFF", in2 := 2)
      wire#w3
      R_Coil( "TRANSFER DB"."PREMIXING VACCUM PUMP MOTOR-W 1 BIT" )
   END_RUNG
   RUNG wire#w2
      Contact( "MANUAL INTERLOCK DB"."MAIN ERROR" )
   END_RUNG wire#w3
   RUNG wire#w2
      Contact( "DI MAPING"."VACCUM PUMP MOTOR 1 TRIP" )
   END_RUNG wire#w3
   RUNG wire#w2
      { S7_Templates := "SrcType := Int" } NE_Contact(in1 := "MANUAL INTERLOCK DB"."PREMIXING TRANSFER PROCESS INTERLOCK", in2 := 2)
   END_RUNG wire#w3
   RUNG wire#w2
      { S7_Templates := "SrcType := Int" } NE_Contact(in1 := "RECIRCULATION DB".PREMIXING.BUFF, in2 := 0)
   END_RUNG wire#w3
   // the same network as SCL:
   IF ("MODE SELECTION DB"."MODE BUFF" <> 2) OR "MANUAL INTERLOCK DB"."MAIN ERROR" OR "DI MAPING"."VACCUM PUMP MOTOR 1 TRIP" OR ("MANUAL INTERLOCK DB"."MFG TRANSFER PROCESS INTERLOCK" <> 2) OR ("RECIRCULATION DB".MFG.BUFF <> 0) THEN
       "TRANSFER DB"."MFG VACCUM PUMP MOTOR-W 1 BIT" := FALSE;
   END_IF;
   IF "AlwaysTRUE" AND (("MODE SELECTION DB"."MODE BUFF" <> 2) OR "MANUAL INTERLOCK DB"."MAIN ERROR" OR "DI MAPING"."VACCUM PUMP MOTOR 1 TRIP" OR ("MANUAL INTERLOCK DB"."PREMIXING TRANSFER PROCESS INTERLOCK" <> 2) OR ("RECIRCULATION DB".PREMIXING.BUFF <> 0)) THEN
       "TRANSFER DB"."PREMIXING VACCUM PUMP MOTOR-W 1 BIT" := FALSE;
   END_IF;
END_REGION

REGION Network 35: VACCUMP PUMP MOTOR 2 RUN
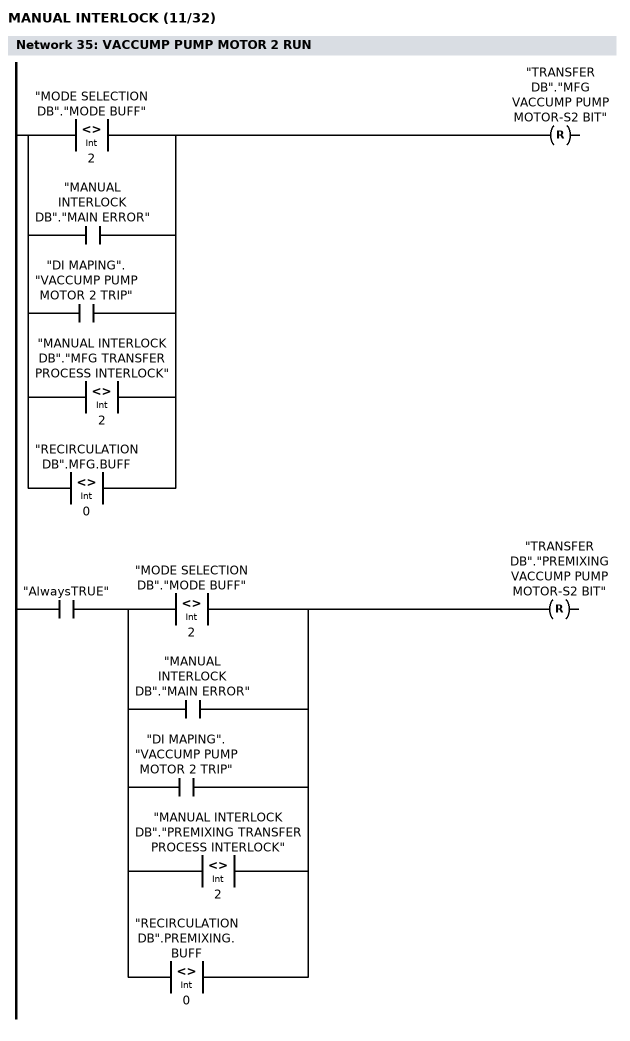
   RUNG wire#powerrail
      { S7_Templates := "SrcType := Int" } NE_Contact(in1 := "MODE SELECTION DB"."MODE BUFF", in2 := 2)
      wire#w1
      R_Coil( "TRANSFER DB"."MFG VACCUMP PUMP MOTOR-S2 BIT" )
   END_RUNG
   RUNG wire#powerrail
      Contact( "MANUAL INTERLOCK DB"."MAIN ERROR" )
   END_RUNG wire#w1
   RUNG wire#powerrail
      Contact( "DI MAPING"."VACCUMP PUMP MOTOR 2 TRIP" )
   END_RUNG wire#w1
   RUNG wire#powerrail
      { S7_Templates := "SrcType := Int" } NE_Contact(in1 := "MANUAL INTERLOCK DB"."MFG TRANSFER PROCESS INTERLOCK", in2 := 2)
   END_RUNG wire#w1
   RUNG wire#powerrail
      { S7_Templates := "SrcType := Int" } NE_Contact(in1 := "RECIRCULATION DB".MFG.BUFF, in2 := 0)
   END_RUNG wire#w1
   RUNG wire#powerrail
      Contact( "AlwaysTRUE" )
      wire#w2
      { S7_Templates := "SrcType := Int" } NE_Contact(in1 := "MODE SELECTION DB"."MODE BUFF", in2 := 2)
      wire#w3
      R_Coil( "TRANSFER DB"."PREMIXING VACCUMP PUMP MOTOR-S2 BIT" )
   END_RUNG
   RUNG wire#w2
      Contact( "MANUAL INTERLOCK DB"."MAIN ERROR" )
   END_RUNG wire#w3
   RUNG wire#w2
      Contact( "DI MAPING"."VACCUMP PUMP MOTOR 2 TRIP" )
   END_RUNG wire#w3
   RUNG wire#w2
      { S7_Templates := "SrcType := Int" } NE_Contact(in1 := "MANUAL INTERLOCK DB"."PREMIXING TRANSFER PROCESS INTERLOCK", in2 := 2)
   END_RUNG wire#w3
   RUNG wire#w2
      { S7_Templates := "SrcType := Int" } NE_Contact(in1 := "RECIRCULATION DB".PREMIXING.BUFF, in2 := 0)
   END_RUNG wire#w3
   // the same network as SCL:
   IF ("MODE SELECTION DB"."MODE BUFF" <> 2) OR "MANUAL INTERLOCK DB"."MAIN ERROR" OR "DI MAPING"."VACCUMP PUMP MOTOR 2 TRIP" OR ("MANUAL INTERLOCK DB"."MFG TRANSFER PROCESS INTERLOCK" <> 2) OR ("RECIRCULATION DB".MFG.BUFF <> 0) THEN
       "TRANSFER DB"."MFG VACCUMP PUMP MOTOR-S2 BIT" := FALSE;
   END_IF;
   IF "AlwaysTRUE" AND (("MODE SELECTION DB"."MODE BUFF" <> 2) OR "MANUAL INTERLOCK DB"."MAIN ERROR" OR "DI MAPING"."VACCUMP PUMP MOTOR 2 TRIP" OR ("MANUAL INTERLOCK DB"."PREMIXING TRANSFER PROCESS INTERLOCK" <> 2) OR ("RECIRCULATION DB".PREMIXING.BUFF <> 0)) THEN
       "TRANSFER DB"."PREMIXING VACCUMP PUMP MOTOR-S2 BIT" := FALSE;
   END_IF;
END_REGION

REGION Network 36: VACCUMP PUMP MOTOR 3 RUN
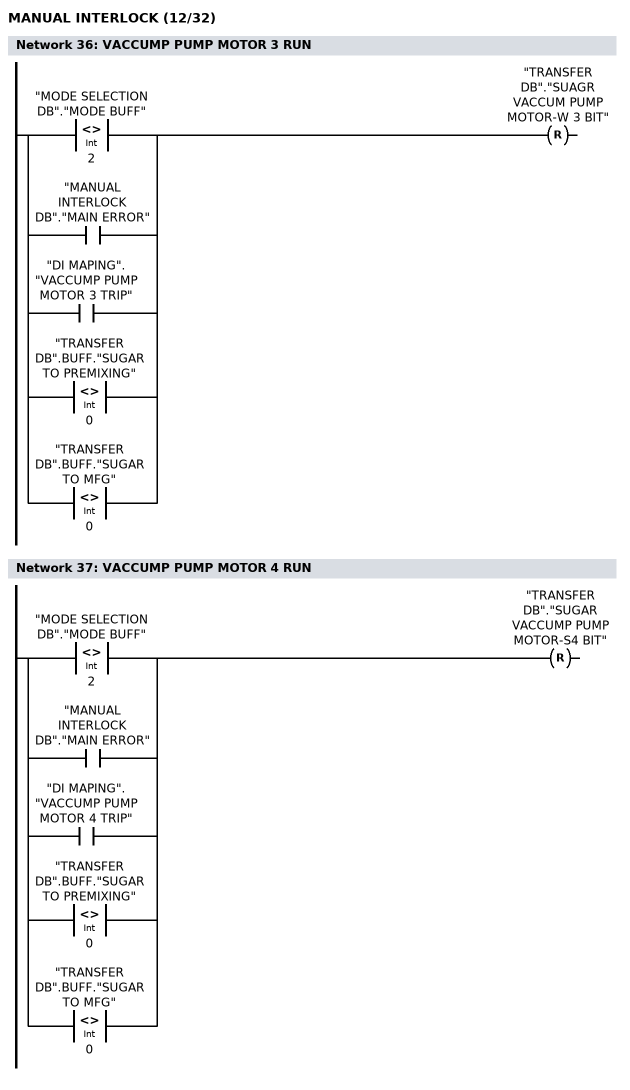
   RUNG wire#powerrail
      { S7_Templates := "SrcType := Int" } NE_Contact(in1 := "MODE SELECTION DB"."MODE BUFF", in2 := 2)
      wire#w1
      R_Coil( "TRANSFER DB"."SUAGR VACCUM PUMP MOTOR-W 3 BIT" )
   END_RUNG
   RUNG wire#powerrail
      Contact( "MANUAL INTERLOCK DB"."MAIN ERROR" )
   END_RUNG wire#w1
   RUNG wire#powerrail
      Contact( "DI MAPING"."VACCUMP PUMP MOTOR 3 TRIP" )
   END_RUNG wire#w1
   RUNG wire#powerrail
      { S7_Templates := "SrcType := Int" } NE_Contact(in1 := "TRANSFER DB".BUFF."SUGAR TO PREMIXING", in2 := 0)
   END_RUNG wire#w1
   RUNG wire#powerrail
      { S7_Templates := "SrcType := Int" } NE_Contact(in1 := "TRANSFER DB".BUFF."SUGAR TO MFG", in2 := 0)
   END_RUNG wire#w1
   // the same network as SCL:
   IF ("MODE SELECTION DB"."MODE BUFF" <> 2) OR "MANUAL INTERLOCK DB"."MAIN ERROR" OR "DI MAPING"."VACCUMP PUMP MOTOR 3 TRIP" OR ("TRANSFER DB".BUFF."SUGAR TO PREMIXING" <> 0) OR ("TRANSFER DB".BUFF."SUGAR TO MFG" <> 0) THEN
       "TRANSFER DB"."SUAGR VACCUM PUMP MOTOR-W 3 BIT" := FALSE;
   END_IF;
END_REGION

REGION Network 37: VACCUMP PUMP MOTOR 4 RUN
   RUNG wire#powerrail
      { S7_Templates := "SrcType := Int" } NE_Contact(in1 := "MODE SELECTION DB"."MODE BUFF", in2 := 2)
      wire#w1
      R_Coil( "TRANSFER DB"."SUGAR VACCUMP PUMP MOTOR-S4 BIT" )
   END_RUNG
   RUNG wire#powerrail
      Contact( "MANUAL INTERLOCK DB"."MAIN ERROR" )
   END_RUNG wire#w1
   RUNG wire#powerrail
      Contact( "DI MAPING"."VACCUMP PUMP MOTOR 4 TRIP" )
   END_RUNG wire#w1
   RUNG wire#powerrail
      { S7_Templates := "SrcType := Int" } NE_Contact(in1 := "TRANSFER DB".BUFF."SUGAR TO PREMIXING", in2 := 0)
   END_RUNG wire#w1
   RUNG wire#powerrail
      { S7_Templates := "SrcType := Int" } NE_Contact(in1 := "TRANSFER DB".BUFF."SUGAR TO MFG", in2 := 0)
   END_RUNG wire#w1
   // the same network as SCL:
   IF ("MODE SELECTION DB"."MODE BUFF" <> 2) OR "MANUAL INTERLOCK DB"."MAIN ERROR" OR "DI MAPING"."VACCUMP PUMP MOTOR 4 TRIP" OR ("TRANSFER DB".BUFF."SUGAR TO PREMIXING" <> 0) OR ("TRANSFER DB".BUFF."SUGAR TO MFG" <> 0) THEN
       "TRANSFER DB"."SUGAR VACCUMP PUMP MOTOR-S4 BIT" := FALSE;
   END_IF;
END_REGION

REGION Network 38: SUGAR VESSEL BOTTOM STERROR RUN
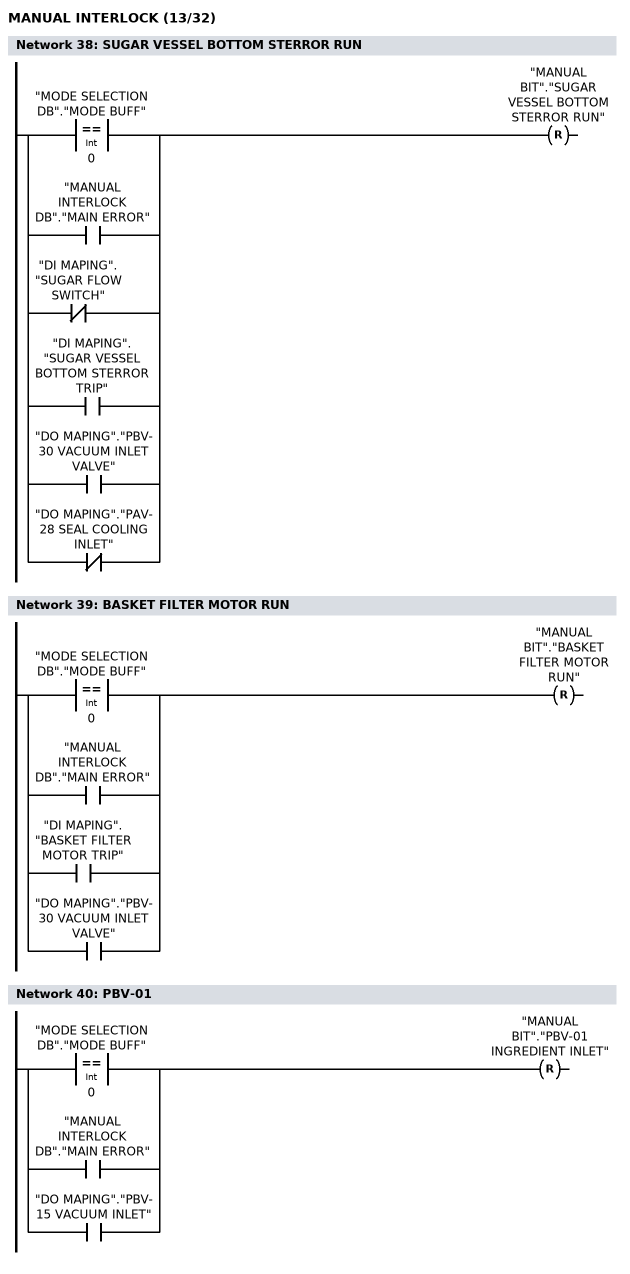
   RUNG wire#powerrail
      { S7_Templates := "SrcType := Int" } EQ_Contact(in1 := "MODE SELECTION DB"."MODE BUFF", in2 := 0)
      wire#w1
      R_Coil( "MANUAL BIT"."SUGAR VESSEL BOTTOM STERROR RUN" )
   END_RUNG
   RUNG wire#powerrail
      Contact( "MANUAL INTERLOCK DB"."MAIN ERROR" )
   END_RUNG wire#w1
   RUNG wire#powerrail
      I_Contact( "DI MAPING"."SUGAR FLOW SWITCH" )
   END_RUNG wire#w1
   RUNG wire#powerrail
      Contact( "DI MAPING"."SUGAR VESSEL BOTTOM STERROR TRIP" )
   END_RUNG wire#w1
   RUNG wire#powerrail
      Contact( "DO MAPING"."PBV-30 VACUUM INLET VALVE" )
   END_RUNG wire#w1
   RUNG wire#powerrail
      I_Contact( "DO MAPING"."PAV-28 SEAL COOLING INLET" )
   END_RUNG wire#w1
   // the same network as SCL:
   IF ("MODE SELECTION DB"."MODE BUFF" = 0) OR "MANUAL INTERLOCK DB"."MAIN ERROR" OR NOT "DI MAPING"."SUGAR FLOW SWITCH" OR "DI MAPING"."SUGAR VESSEL BOTTOM STERROR TRIP" OR "DO MAPING"."PBV-30 VACUUM INLET VALVE" OR NOT "DO MAPING"."PAV-28 SEAL COOLING INLET" THEN
       "MANUAL BIT"."SUGAR VESSEL BOTTOM STERROR RUN" := FALSE;
   END_IF;
END_REGION

REGION Network 39: BASKET FILTER MOTOR RUN
   RUNG wire#powerrail
      { S7_Templates := "SrcType := Int" } EQ_Contact(in1 := "MODE SELECTION DB"."MODE BUFF", in2 := 0)
      wire#w1
      R_Coil( "MANUAL BIT"."BASKET FILTER MOTOR RUN" )
   END_RUNG
   RUNG wire#powerrail
      Contact( "MANUAL INTERLOCK DB"."MAIN ERROR" )
   END_RUNG wire#w1
   RUNG wire#powerrail
      Contact( "DI MAPING"."BASKET FILTER MOTOR TRIP" )
   END_RUNG wire#w1
   RUNG wire#powerrail
      Contact( "DO MAPING"."PBV-30 VACUUM INLET VALVE" )
   END_RUNG wire#w1
   // the same network as SCL:
   IF ("MODE SELECTION DB"."MODE BUFF" = 0) OR "MANUAL INTERLOCK DB"."MAIN ERROR" OR "DI MAPING"."BASKET FILTER MOTOR TRIP" OR "DO MAPING"."PBV-30 VACUUM INLET VALVE" THEN
       "MANUAL BIT"."BASKET FILTER MOTOR RUN" := FALSE;
   END_IF;
END_REGION

REGION Network 40: PBV-01
   RUNG wire#powerrail
      { S7_Templates := "SrcType := Int" } EQ_Contact(in1 := "MODE SELECTION DB"."MODE BUFF", in2 := 0)
      wire#w1
      R_Coil( "MANUAL BIT"."PBV-01 INGREDIENT INLET" )
   END_RUNG
   RUNG wire#powerrail
      Contact( "MANUAL INTERLOCK DB"."MAIN ERROR" )
   END_RUNG wire#w1
   RUNG wire#powerrail
      Contact( "DO MAPING"."PBV-15 VACUUM INLET" )
   END_RUNG wire#w1
   // the same network as SCL:
   IF ("MODE SELECTION DB"."MODE BUFF" = 0) OR "MANUAL INTERLOCK DB"."MAIN ERROR" OR "DO MAPING"."PBV-15 VACUUM INLET" THEN
       "MANUAL BIT"."PBV-01 INGREDIENT INLET" := FALSE;
   END_IF;
END_REGION

REGION Network 41: PBV-02
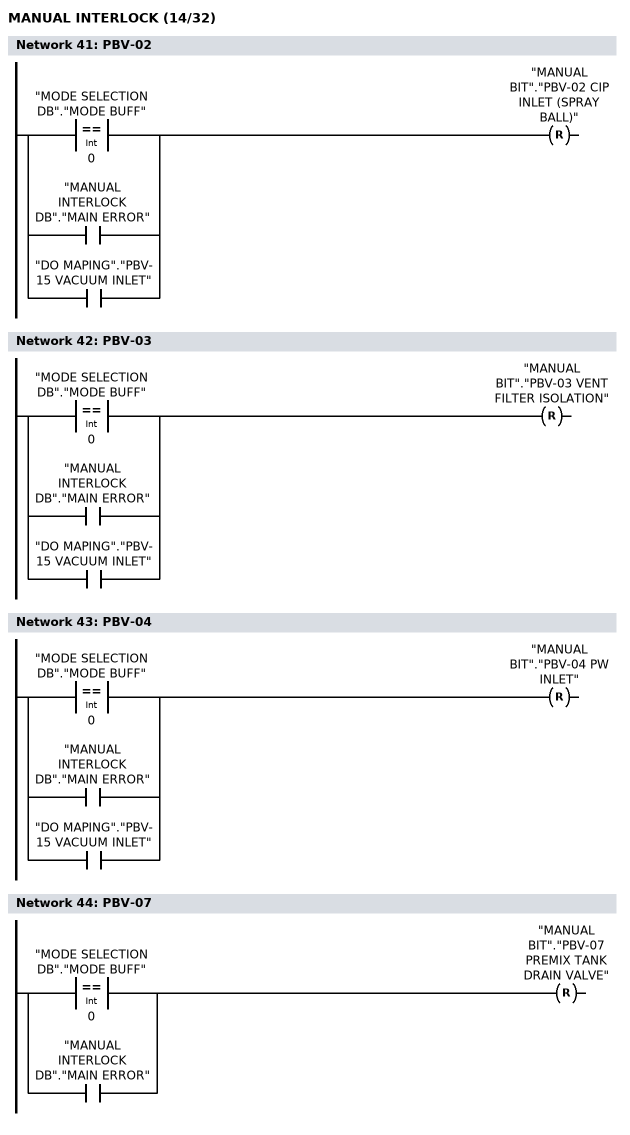
   RUNG wire#powerrail
      { S7_Templates := "SrcType := Int" } EQ_Contact(in1 := "MODE SELECTION DB"."MODE BUFF", in2 := 0)
      wire#w1
      R_Coil( "MANUAL BIT"."PBV-02 CIP INLET (SPRAY BALL)" )
   END_RUNG
   RUNG wire#powerrail
      Contact( "MANUAL INTERLOCK DB"."MAIN ERROR" )
   END_RUNG wire#w1
   RUNG wire#powerrail
      Contact( "DO MAPING"."PBV-15 VACUUM INLET" )
   END_RUNG wire#w1
   // the same network as SCL:
   IF ("MODE SELECTION DB"."MODE BUFF" = 0) OR "MANUAL INTERLOCK DB"."MAIN ERROR" OR "DO MAPING"."PBV-15 VACUUM INLET" THEN
       "MANUAL BIT"."PBV-02 CIP INLET (SPRAY BALL)" := FALSE;
   END_IF;
END_REGION

REGION Network 42: PBV-03
   RUNG wire#powerrail
      { S7_Templates := "SrcType := Int" } EQ_Contact(in1 := "MODE SELECTION DB"."MODE BUFF", in2 := 0)
      wire#w1
      R_Coil( "MANUAL BIT"."PBV-03 VENT FILTER ISOLATION" )
   END_RUNG
   RUNG wire#powerrail
      Contact( "MANUAL INTERLOCK DB"."MAIN ERROR" )
   END_RUNG wire#w1
   RUNG wire#powerrail
      Contact( "DO MAPING"."PBV-15 VACUUM INLET" )
   END_RUNG wire#w1
   // the same network as SCL:
   IF ("MODE SELECTION DB"."MODE BUFF" = 0) OR "MANUAL INTERLOCK DB"."MAIN ERROR" OR "DO MAPING"."PBV-15 VACUUM INLET" THEN
       "MANUAL BIT"."PBV-03 VENT FILTER ISOLATION" := FALSE;
   END_IF;
END_REGION

REGION Network 43: PBV-04
   RUNG wire#powerrail
      { S7_Templates := "SrcType := Int" } EQ_Contact(in1 := "MODE SELECTION DB"."MODE BUFF", in2 := 0)
      wire#w1
      R_Coil( "MANUAL BIT"."PBV-04 PW INLET" )
   END_RUNG
   RUNG wire#powerrail
      Contact( "MANUAL INTERLOCK DB"."MAIN ERROR" )
   END_RUNG wire#w1
   RUNG wire#powerrail
      Contact( "DO MAPING"."PBV-15 VACUUM INLET" )
   END_RUNG wire#w1
   // the same network as SCL:
   IF ("MODE SELECTION DB"."MODE BUFF" = 0) OR "MANUAL INTERLOCK DB"."MAIN ERROR" OR "DO MAPING"."PBV-15 VACUUM INLET" THEN
       "MANUAL BIT"."PBV-04 PW INLET" := FALSE;
   END_IF;
END_REGION

REGION Network 44: PBV-07
   RUNG wire#powerrail
      { S7_Templates := "SrcType := Int" } EQ_Contact(in1 := "MODE SELECTION DB"."MODE BUFF", in2 := 0)
      wire#w1
      R_Coil( "MANUAL BIT"."PBV-07 PREMIX TANK DRAIN VALVE" )
   END_RUNG
   RUNG wire#powerrail
      Contact( "MANUAL INTERLOCK DB"."MAIN ERROR" )
   END_RUNG wire#w1
   // the same network as SCL:
   IF ("MODE SELECTION DB"."MODE BUFF" = 0) OR "MANUAL INTERLOCK DB"."MAIN ERROR" THEN
       "MANUAL BIT"."PBV-07 PREMIX TANK DRAIN VALVE" := FALSE;
   END_IF;
END_REGION

REGION Network 45: PAV-09
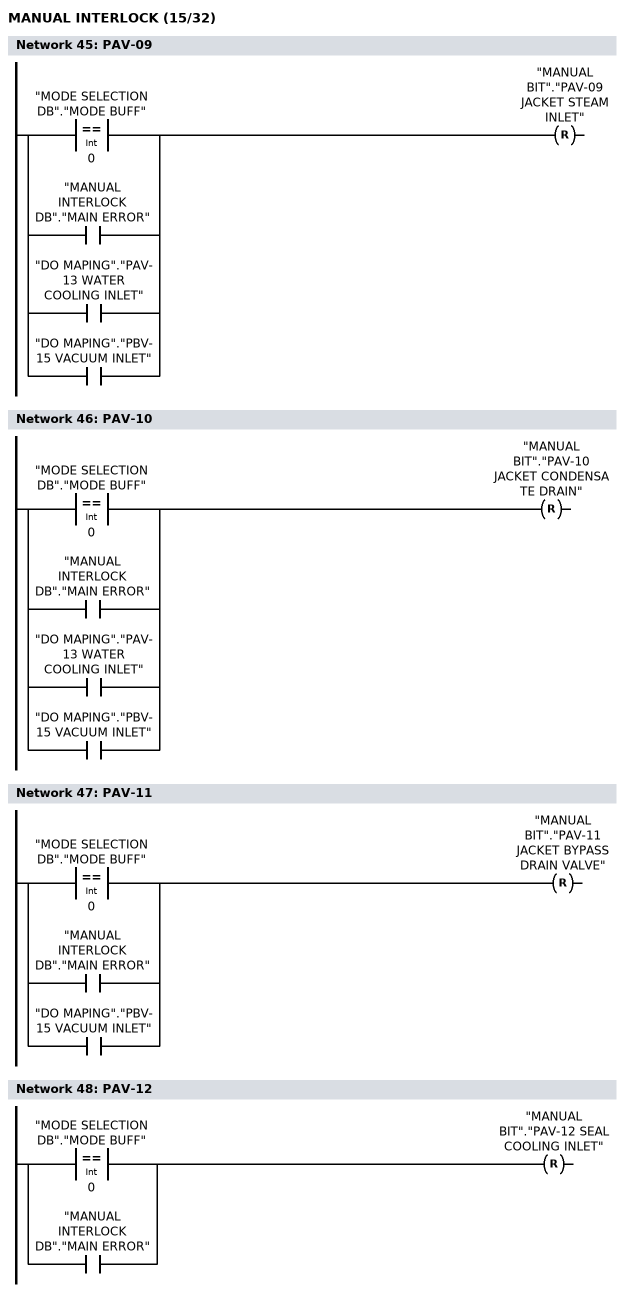
   RUNG wire#powerrail
      { S7_Templates := "SrcType := Int" } EQ_Contact(in1 := "MODE SELECTION DB"."MODE BUFF", in2 := 0)
      wire#w1
      R_Coil( "MANUAL BIT"."PAV-09 JACKET STEAM INLET" )
   END_RUNG
   RUNG wire#powerrail
      Contact( "MANUAL INTERLOCK DB"."MAIN ERROR" )
   END_RUNG wire#w1
   RUNG wire#powerrail
      Contact( "DO MAPING"."PAV-13 WATER COOLING INLET" )
   END_RUNG wire#w1
   RUNG wire#powerrail
      Contact( "DO MAPING"."PBV-15 VACUUM INLET" )
   END_RUNG wire#w1
   // the same network as SCL:
   IF ("MODE SELECTION DB"."MODE BUFF" = 0) OR "MANUAL INTERLOCK DB"."MAIN ERROR" OR "DO MAPING"."PAV-13 WATER COOLING INLET" OR "DO MAPING"."PBV-15 VACUUM INLET" THEN
       "MANUAL BIT"."PAV-09 JACKET STEAM INLET" := FALSE;
   END_IF;
END_REGION

REGION Network 46: PAV-10
   RUNG wire#powerrail
      { S7_Templates := "SrcType := Int" } EQ_Contact(in1 := "MODE SELECTION DB"."MODE BUFF", in2 := 0)
      wire#w1
      R_Coil( "MANUAL BIT"."PAV-10 JACKET CONDENSATE DRAIN" )
   END_RUNG
   RUNG wire#powerrail
      Contact( "MANUAL INTERLOCK DB"."MAIN ERROR" )
   END_RUNG wire#w1
   RUNG wire#powerrail
      Contact( "DO MAPING"."PAV-13 WATER COOLING INLET" )
   END_RUNG wire#w1
   RUNG wire#powerrail
      Contact( "DO MAPING"."PBV-15 VACUUM INLET" )
   END_RUNG wire#w1
   // the same network as SCL:
   IF ("MODE SELECTION DB"."MODE BUFF" = 0) OR "MANUAL INTERLOCK DB"."MAIN ERROR" OR "DO MAPING"."PAV-13 WATER COOLING INLET" OR "DO MAPING"."PBV-15 VACUUM INLET" THEN
       "MANUAL BIT"."PAV-10 JACKET CONDENSATE DRAIN" := FALSE;
   END_IF;
END_REGION

REGION Network 47: PAV-11
   RUNG wire#powerrail
      { S7_Templates := "SrcType := Int" } EQ_Contact(in1 := "MODE SELECTION DB"."MODE BUFF", in2 := 0)
      wire#w1
      R_Coil( "MANUAL BIT"."PAV-11 JACKET BYPASS DRAIN VALVE" )
   END_RUNG
   RUNG wire#powerrail
      Contact( "MANUAL INTERLOCK DB"."MAIN ERROR" )
   END_RUNG wire#w1
   RUNG wire#powerrail
      Contact( "DO MAPING"."PBV-15 VACUUM INLET" )
   END_RUNG wire#w1
   // the same network as SCL:
   IF ("MODE SELECTION DB"."MODE BUFF" = 0) OR "MANUAL INTERLOCK DB"."MAIN ERROR" OR "DO MAPING"."PBV-15 VACUUM INLET" THEN
       "MANUAL BIT"."PAV-11 JACKET BYPASS DRAIN VALVE" := FALSE;
   END_IF;
END_REGION

REGION Network 48: PAV-12
   RUNG wire#powerrail
      { S7_Templates := "SrcType := Int" } EQ_Contact(in1 := "MODE SELECTION DB"."MODE BUFF", in2 := 0)
      wire#w1
      R_Coil( "MANUAL BIT"."PAV-12 SEAL COOLING INLET" )
   END_RUNG
   RUNG wire#powerrail
      Contact( "MANUAL INTERLOCK DB"."MAIN ERROR" )
   END_RUNG wire#w1
   // the same network as SCL:
   IF ("MODE SELECTION DB"."MODE BUFF" = 0) OR "MANUAL INTERLOCK DB"."MAIN ERROR" THEN
       "MANUAL BIT"."PAV-12 SEAL COOLING INLET" := FALSE;
   END_IF;
END_REGION

REGION Network 49: PAV-13
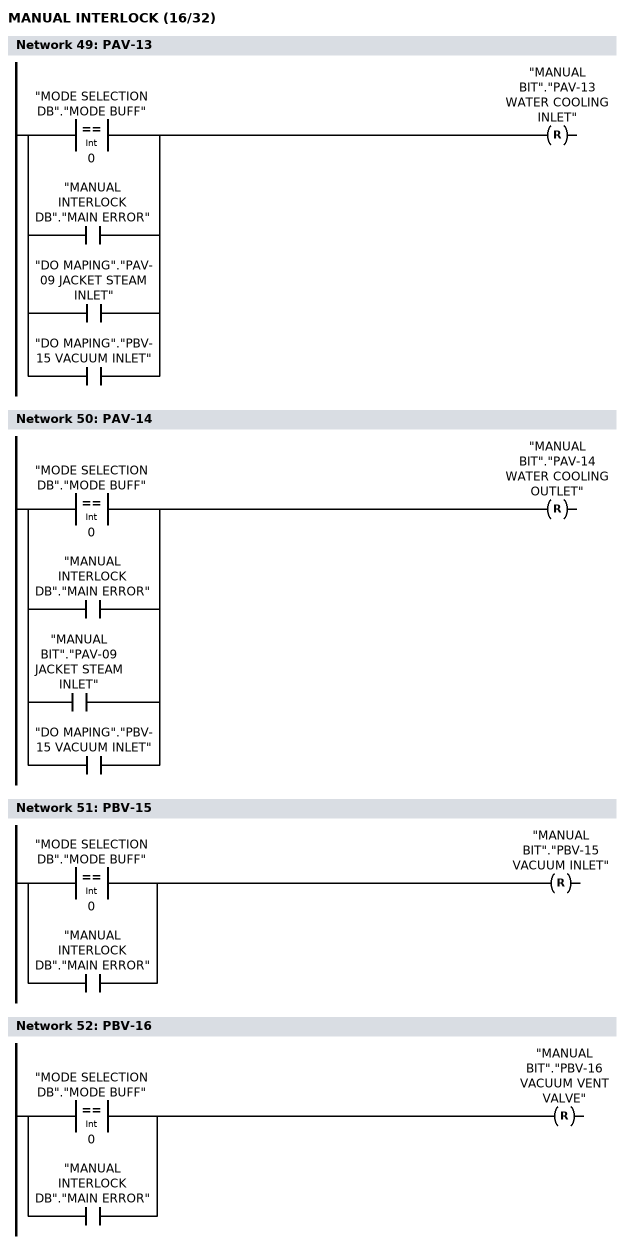
   RUNG wire#powerrail
      { S7_Templates := "SrcType := Int" } EQ_Contact(in1 := "MODE SELECTION DB"."MODE BUFF", in2 := 0)
      wire#w1
      R_Coil( "MANUAL BIT"."PAV-13 WATER COOLING INLET" )
   END_RUNG
   RUNG wire#powerrail
      Contact( "MANUAL INTERLOCK DB"."MAIN ERROR" )
   END_RUNG wire#w1
   RUNG wire#powerrail
      Contact( "DO MAPING"."PAV-09 JACKET STEAM INLET" )
   END_RUNG wire#w1
   RUNG wire#powerrail
      Contact( "DO MAPING"."PBV-15 VACUUM INLET" )
   END_RUNG wire#w1
   // the same network as SCL:
   IF ("MODE SELECTION DB"."MODE BUFF" = 0) OR "MANUAL INTERLOCK DB"."MAIN ERROR" OR "DO MAPING"."PAV-09 JACKET STEAM INLET" OR "DO MAPING"."PBV-15 VACUUM INLET" THEN
       "MANUAL BIT"."PAV-13 WATER COOLING INLET" := FALSE;
   END_IF;
END_REGION

REGION Network 50: PAV-14
   RUNG wire#powerrail
      { S7_Templates := "SrcType := Int" } EQ_Contact(in1 := "MODE SELECTION DB"."MODE BUFF", in2 := 0)
      wire#w1
      R_Coil( "MANUAL BIT"."PAV-14 WATER COOLING OUTLET" )
   END_RUNG
   RUNG wire#powerrail
      Contact( "MANUAL INTERLOCK DB"."MAIN ERROR" )
   END_RUNG wire#w1
   RUNG wire#powerrail
      Contact( "MANUAL BIT"."PAV-09 JACKET STEAM INLET" )
   END_RUNG wire#w1
   RUNG wire#powerrail
      Contact( "DO MAPING"."PBV-15 VACUUM INLET" )
   END_RUNG wire#w1
   // the same network as SCL:
   IF ("MODE SELECTION DB"."MODE BUFF" = 0) OR "MANUAL INTERLOCK DB"."MAIN ERROR" OR "MANUAL BIT"."PAV-09 JACKET STEAM INLET" OR "DO MAPING"."PBV-15 VACUUM INLET" THEN
       "MANUAL BIT"."PAV-14 WATER COOLING OUTLET" := FALSE;
   END_IF;
END_REGION

REGION Network 51: PBV-15
   RUNG wire#powerrail
      { S7_Templates := "SrcType := Int" } EQ_Contact(in1 := "MODE SELECTION DB"."MODE BUFF", in2 := 0)
      wire#w1
      R_Coil( "MANUAL BIT"."PBV-15 VACUUM INLET" )
   END_RUNG
   RUNG wire#powerrail
      Contact( "MANUAL INTERLOCK DB"."MAIN ERROR" )
   END_RUNG wire#w1
   // the same network as SCL:
   IF ("MODE SELECTION DB"."MODE BUFF" = 0) OR "MANUAL INTERLOCK DB"."MAIN ERROR" THEN
       "MANUAL BIT"."PBV-15 VACUUM INLET" := FALSE;
   END_IF;
END_REGION

REGION Network 52: PBV-16
   RUNG wire#powerrail
      { S7_Templates := "SrcType := Int" } EQ_Contact(in1 := "MODE SELECTION DB"."MODE BUFF", in2 := 0)
      wire#w1
      R_Coil( "MANUAL BIT"."PBV-16 VACUUM VENT VALVE" )
   END_RUNG
   RUNG wire#powerrail
      Contact( "MANUAL INTERLOCK DB"."MAIN ERROR" )
   END_RUNG wire#w1
   // the same network as SCL:
   IF ("MODE SELECTION DB"."MODE BUFF" = 0) OR "MANUAL INTERLOCK DB"."MAIN ERROR" THEN
       "MANUAL BIT"."PBV-16 VACUUM VENT VALVE" := FALSE;
   END_IF;
END_REGION

REGION Network 53: PFBV-17
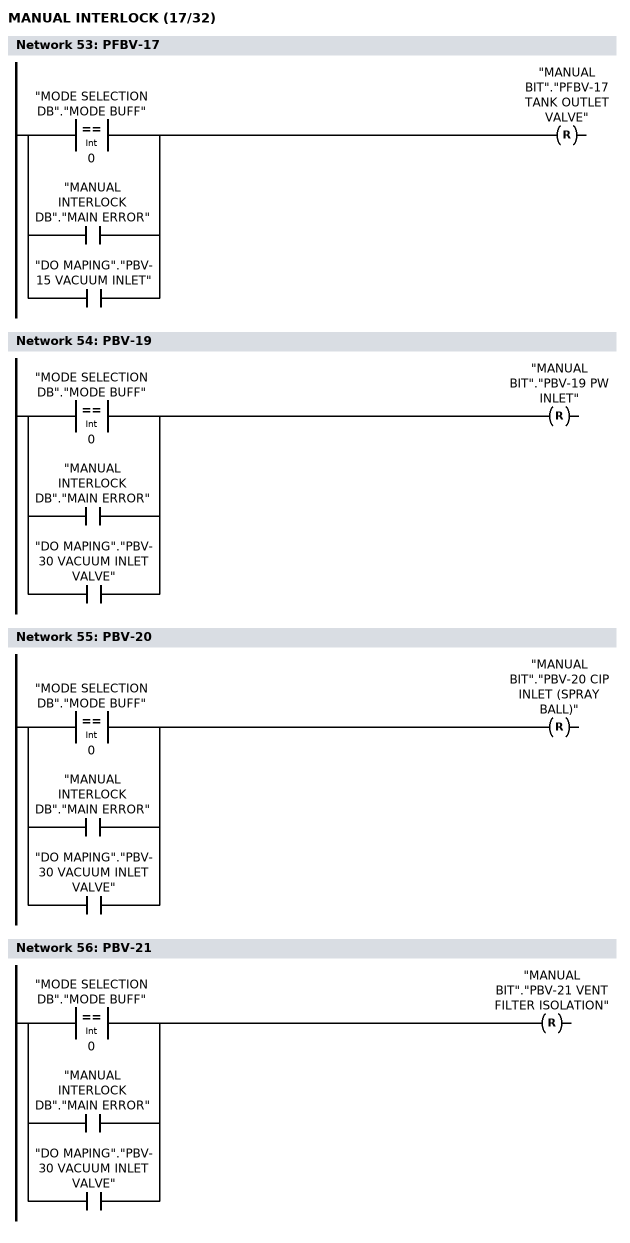
   RUNG wire#powerrail
      { S7_Templates := "SrcType := Int" } EQ_Contact(in1 := "MODE SELECTION DB"."MODE BUFF", in2 := 0)
      wire#w1
      R_Coil( "MANUAL BIT"."PFBV-17 TANK OUTLET VALVE" )
   END_RUNG
   RUNG wire#powerrail
      Contact( "MANUAL INTERLOCK DB"."MAIN ERROR" )
   END_RUNG wire#w1
   RUNG wire#powerrail
      Contact( "DO MAPING"."PBV-15 VACUUM INLET" )
   END_RUNG wire#w1
   // the same network as SCL:
   IF ("MODE SELECTION DB"."MODE BUFF" = 0) OR "MANUAL INTERLOCK DB"."MAIN ERROR" OR "DO MAPING"."PBV-15 VACUUM INLET" THEN
       "MANUAL BIT"."PFBV-17 TANK OUTLET VALVE" := FALSE;
   END_IF;
END_REGION

REGION Network 54: PBV-19
   RUNG wire#powerrail
      { S7_Templates := "SrcType := Int" } EQ_Contact(in1 := "MODE SELECTION DB"."MODE BUFF", in2 := 0)
      wire#w1
      R_Coil( "MANUAL BIT"."PBV-19 PW INLET" )
   END_RUNG
   RUNG wire#powerrail
      Contact( "MANUAL INTERLOCK DB"."MAIN ERROR" )
   END_RUNG wire#w1
   RUNG wire#powerrail
      Contact( "DO MAPING"."PBV-30 VACUUM INLET VALVE" )
   END_RUNG wire#w1
   // the same network as SCL:
   IF ("MODE SELECTION DB"."MODE BUFF" = 0) OR "MANUAL INTERLOCK DB"."MAIN ERROR" OR "DO MAPING"."PBV-30 VACUUM INLET VALVE" THEN
       "MANUAL BIT"."PBV-19 PW INLET" := FALSE;
   END_IF;
END_REGION

REGION Network 55: PBV-20
   RUNG wire#powerrail
      { S7_Templates := "SrcType := Int" } EQ_Contact(in1 := "MODE SELECTION DB"."MODE BUFF", in2 := 0)
      wire#w1
      R_Coil( "MANUAL BIT"."PBV-20 CIP INLET (SPRAY BALL)" )
   END_RUNG
   RUNG wire#powerrail
      Contact( "MANUAL INTERLOCK DB"."MAIN ERROR" )
   END_RUNG wire#w1
   RUNG wire#powerrail
      Contact( "DO MAPING"."PBV-30 VACUUM INLET VALVE" )
   END_RUNG wire#w1
   // the same network as SCL:
   IF ("MODE SELECTION DB"."MODE BUFF" = 0) OR "MANUAL INTERLOCK DB"."MAIN ERROR" OR "DO MAPING"."PBV-30 VACUUM INLET VALVE" THEN
       "MANUAL BIT"."PBV-20 CIP INLET (SPRAY BALL)" := FALSE;
   END_IF;
END_REGION

REGION Network 56: PBV-21
   RUNG wire#powerrail
      { S7_Templates := "SrcType := Int" } EQ_Contact(in1 := "MODE SELECTION DB"."MODE BUFF", in2 := 0)
      wire#w1
      R_Coil( "MANUAL BIT"."PBV-21 VENT FILTER ISOLATION" )
   END_RUNG
   RUNG wire#powerrail
      Contact( "MANUAL INTERLOCK DB"."MAIN ERROR" )
   END_RUNG wire#w1
   RUNG wire#powerrail
      Contact( "DO MAPING"."PBV-30 VACUUM INLET VALVE" )
   END_RUNG wire#w1
   // the same network as SCL:
   IF ("MODE SELECTION DB"."MODE BUFF" = 0) OR "MANUAL INTERLOCK DB"."MAIN ERROR" OR "DO MAPING"."PBV-30 VACUUM INLET VALVE" THEN
       "MANUAL BIT"."PBV-21 VENT FILTER ISOLATION" := FALSE;
   END_IF;
END_REGION

REGION Network 57: PBV-22
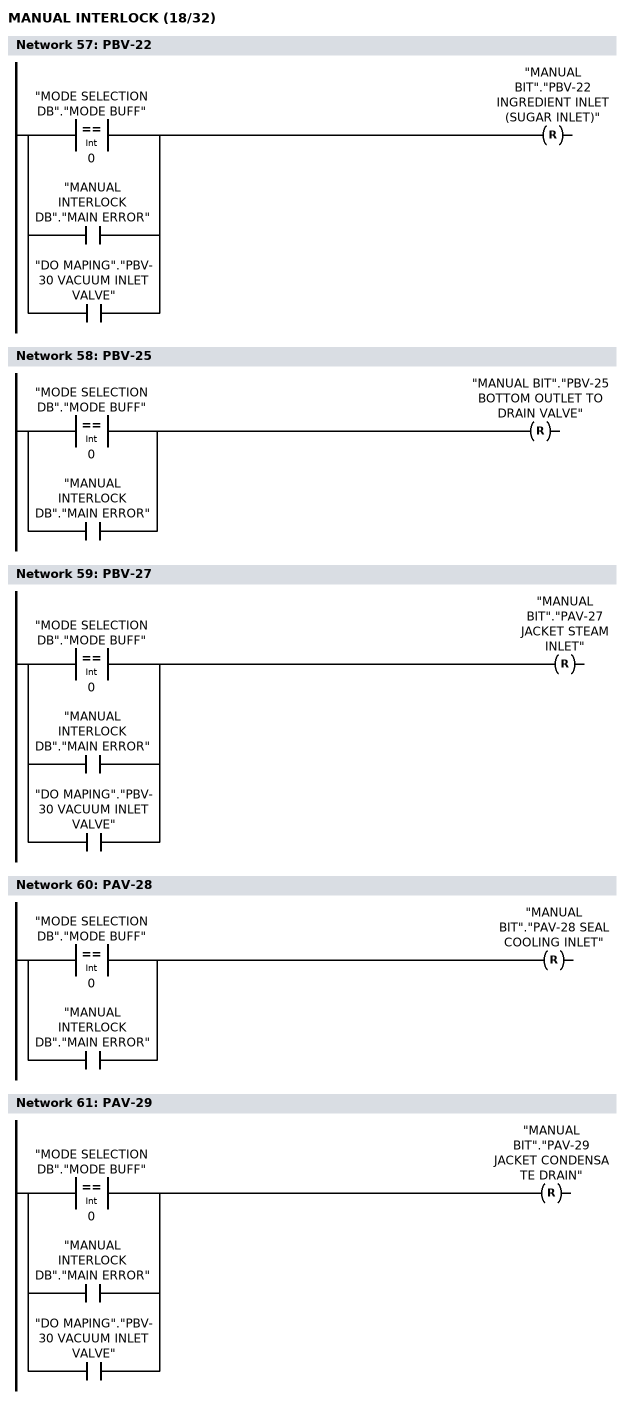
   RUNG wire#powerrail
      { S7_Templates := "SrcType := Int" } EQ_Contact(in1 := "MODE SELECTION DB"."MODE BUFF", in2 := 0)
      wire#w1
      R_Coil( "MANUAL BIT"."PBV-22 INGREDIENT INLET (SUGAR INLET)" )
   END_RUNG
   RUNG wire#powerrail
      Contact( "MANUAL INTERLOCK DB"."MAIN ERROR" )
   END_RUNG wire#w1
   RUNG wire#powerrail
      Contact( "DO MAPING"."PBV-30 VACUUM INLET VALVE" )
   END_RUNG wire#w1
   // the same network as SCL:
   IF ("MODE SELECTION DB"."MODE BUFF" = 0) OR "MANUAL INTERLOCK DB"."MAIN ERROR" OR "DO MAPING"."PBV-30 VACUUM INLET VALVE" THEN
       "MANUAL BIT"."PBV-22 INGREDIENT INLET (SUGAR INLET)" := FALSE;
   END_IF;
END_REGION

REGION Network 58: PBV-25
   RUNG wire#powerrail
      { S7_Templates := "SrcType := Int" } EQ_Contact(in1 := "MODE SELECTION DB"."MODE BUFF", in2 := 0)
      wire#w1
      R_Coil( "MANUAL BIT"."PBV-25 BOTTOM OUTLET TO DRAIN VALVE" )
   END_RUNG
   RUNG wire#powerrail
      Contact( "MANUAL INTERLOCK DB"."MAIN ERROR" )
   END_RUNG wire#w1
   // the same network as SCL:
   IF ("MODE SELECTION DB"."MODE BUFF" = 0) OR "MANUAL INTERLOCK DB"."MAIN ERROR" THEN
       "MANUAL BIT"."PBV-25 BOTTOM OUTLET TO DRAIN VALVE" := FALSE;
   END_IF;
END_REGION

REGION Network 59: PBV-27
   RUNG wire#powerrail
      { S7_Templates := "SrcType := Int" } EQ_Contact(in1 := "MODE SELECTION DB"."MODE BUFF", in2 := 0)
      wire#w1
      R_Coil( "MANUAL BIT"."PAV-27 JACKET STEAM INLET" )
   END_RUNG
   RUNG wire#powerrail
      Contact( "MANUAL INTERLOCK DB"."MAIN ERROR" )
   END_RUNG wire#w1
   RUNG wire#powerrail
      Contact( "DO MAPING"."PBV-30 VACUUM INLET VALVE" )
   END_RUNG wire#w1
   // the same network as SCL:
   IF ("MODE SELECTION DB"."MODE BUFF" = 0) OR "MANUAL INTERLOCK DB"."MAIN ERROR" OR "DO MAPING"."PBV-30 VACUUM INLET VALVE" THEN
       "MANUAL BIT"."PAV-27 JACKET STEAM INLET" := FALSE;
   END_IF;
END_REGION

REGION Network 60: PAV-28
   RUNG wire#powerrail
      { S7_Templates := "SrcType := Int" } EQ_Contact(in1 := "MODE SELECTION DB"."MODE BUFF", in2 := 0)
      wire#w1
      R_Coil( "MANUAL BIT"."PAV-28 SEAL COOLING INLET" )
   END_RUNG
   RUNG wire#powerrail
      Contact( "MANUAL INTERLOCK DB"."MAIN ERROR" )
   END_RUNG wire#w1
   // the same network as SCL:
   IF ("MODE SELECTION DB"."MODE BUFF" = 0) OR "MANUAL INTERLOCK DB"."MAIN ERROR" THEN
       "MANUAL BIT"."PAV-28 SEAL COOLING INLET" := FALSE;
   END_IF;
END_REGION

REGION Network 61: PAV-29
   RUNG wire#powerrail
      { S7_Templates := "SrcType := Int" } EQ_Contact(in1 := "MODE SELECTION DB"."MODE BUFF", in2 := 0)
      wire#w1
      R_Coil( "MANUAL BIT"."PAV-29 JACKET CONDENSATE DRAIN" )
   END_RUNG
   RUNG wire#powerrail
      Contact( "MANUAL INTERLOCK DB"."MAIN ERROR" )
   END_RUNG wire#w1
   RUNG wire#powerrail
      Contact( "DO MAPING"."PBV-30 VACUUM INLET VALVE" )
   END_RUNG wire#w1
   // the same network as SCL:
   IF ("MODE SELECTION DB"."MODE BUFF" = 0) OR "MANUAL INTERLOCK DB"."MAIN ERROR" OR "DO MAPING"."PBV-30 VACUUM INLET VALVE" THEN
       "MANUAL BIT"."PAV-29 JACKET CONDENSATE DRAIN" := FALSE;
   END_IF;
END_REGION

REGION Network 62: PBV-30
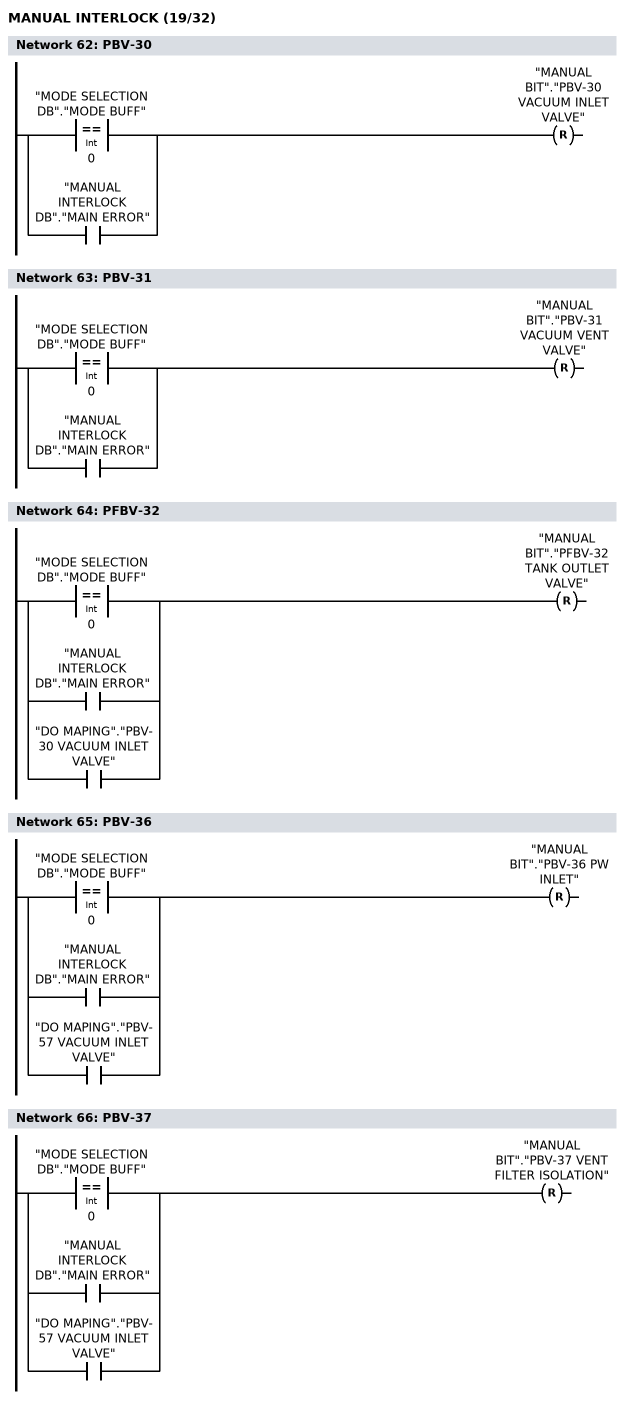
   RUNG wire#powerrail
      { S7_Templates := "SrcType := Int" } EQ_Contact(in1 := "MODE SELECTION DB"."MODE BUFF", in2 := 0)
      wire#w1
      R_Coil( "MANUAL BIT"."PBV-30 VACUUM INLET VALVE" )
   END_RUNG
   RUNG wire#powerrail
      Contact( "MANUAL INTERLOCK DB"."MAIN ERROR" )
   END_RUNG wire#w1
   // the same network as SCL:
   IF ("MODE SELECTION DB"."MODE BUFF" = 0) OR "MANUAL INTERLOCK DB"."MAIN ERROR" THEN
       "MANUAL BIT"."PBV-30 VACUUM INLET VALVE" := FALSE;
   END_IF;
END_REGION

REGION Network 63: PBV-31
   RUNG wire#powerrail
      { S7_Templates := "SrcType := Int" } EQ_Contact(in1 := "MODE SELECTION DB"."MODE BUFF", in2 := 0)
      wire#w1
      R_Coil( "MANUAL BIT"."PBV-31 VACUUM VENT VALVE" )
   END_RUNG
   RUNG wire#powerrail
      Contact( "MANUAL INTERLOCK DB"."MAIN ERROR" )
   END_RUNG wire#w1
   // the same network as SCL:
   IF ("MODE SELECTION DB"."MODE BUFF" = 0) OR "MANUAL INTERLOCK DB"."MAIN ERROR" THEN
       "MANUAL BIT"."PBV-31 VACUUM VENT VALVE" := FALSE;
   END_IF;
END_REGION

REGION Network 64: PFBV-32
   RUNG wire#powerrail
      { S7_Templates := "SrcType := Int" } EQ_Contact(in1 := "MODE SELECTION DB"."MODE BUFF", in2 := 0)
      wire#w1
      R_Coil( "MANUAL BIT"."PFBV-32 TANK OUTLET VALVE" )
   END_RUNG
   RUNG wire#powerrail
      Contact( "MANUAL INTERLOCK DB"."MAIN ERROR" )
   END_RUNG wire#w1
   RUNG wire#powerrail
      Contact( "DO MAPING"."PBV-30 VACUUM INLET VALVE" )
   END_RUNG wire#w1
   // the same network as SCL:
   IF ("MODE SELECTION DB"."MODE BUFF" = 0) OR "MANUAL INTERLOCK DB"."MAIN ERROR" OR "DO MAPING"."PBV-30 VACUUM INLET VALVE" THEN
       "MANUAL BIT"."PFBV-32 TANK OUTLET VALVE" := FALSE;
   END_IF;
END_REGION

REGION Network 65: PBV-36
   RUNG wire#powerrail
      { S7_Templates := "SrcType := Int" } EQ_Contact(in1 := "MODE SELECTION DB"."MODE BUFF", in2 := 0)
      wire#w1
      R_Coil( "MANUAL BIT"."PBV-36 PW INLET" )
   END_RUNG
   RUNG wire#powerrail
      Contact( "MANUAL INTERLOCK DB"."MAIN ERROR" )
   END_RUNG wire#w1
   RUNG wire#powerrail
      Contact( "DO MAPING"."PBV-57 VACUUM INLET VALVE" )
   END_RUNG wire#w1
   // the same network as SCL:
   IF ("MODE SELECTION DB"."MODE BUFF" = 0) OR "MANUAL INTERLOCK DB"."MAIN ERROR" OR "DO MAPING"."PBV-57 VACUUM INLET VALVE" THEN
       "MANUAL BIT"."PBV-36 PW INLET" := FALSE;
   END_IF;
END_REGION

REGION Network 66: PBV-37
   RUNG wire#powerrail
      { S7_Templates := "SrcType := Int" } EQ_Contact(in1 := "MODE SELECTION DB"."MODE BUFF", in2 := 0)
      wire#w1
      R_Coil( "MANUAL BIT"."PBV-37 VENT FILTER ISOLATION" )
   END_RUNG
   RUNG wire#powerrail
      Contact( "MANUAL INTERLOCK DB"."MAIN ERROR" )
   END_RUNG wire#w1
   RUNG wire#powerrail
      Contact( "DO MAPING"."PBV-57 VACUUM INLET VALVE" )
   END_RUNG wire#w1
   // the same network as SCL:
   IF ("MODE SELECTION DB"."MODE BUFF" = 0) OR "MANUAL INTERLOCK DB"."MAIN ERROR" OR "DO MAPING"."PBV-57 VACUUM INLET VALVE" THEN
       "MANUAL BIT"."PBV-37 VENT FILTER ISOLATION" := FALSE;
   END_IF;
END_REGION

REGION Network 67: PBV-38
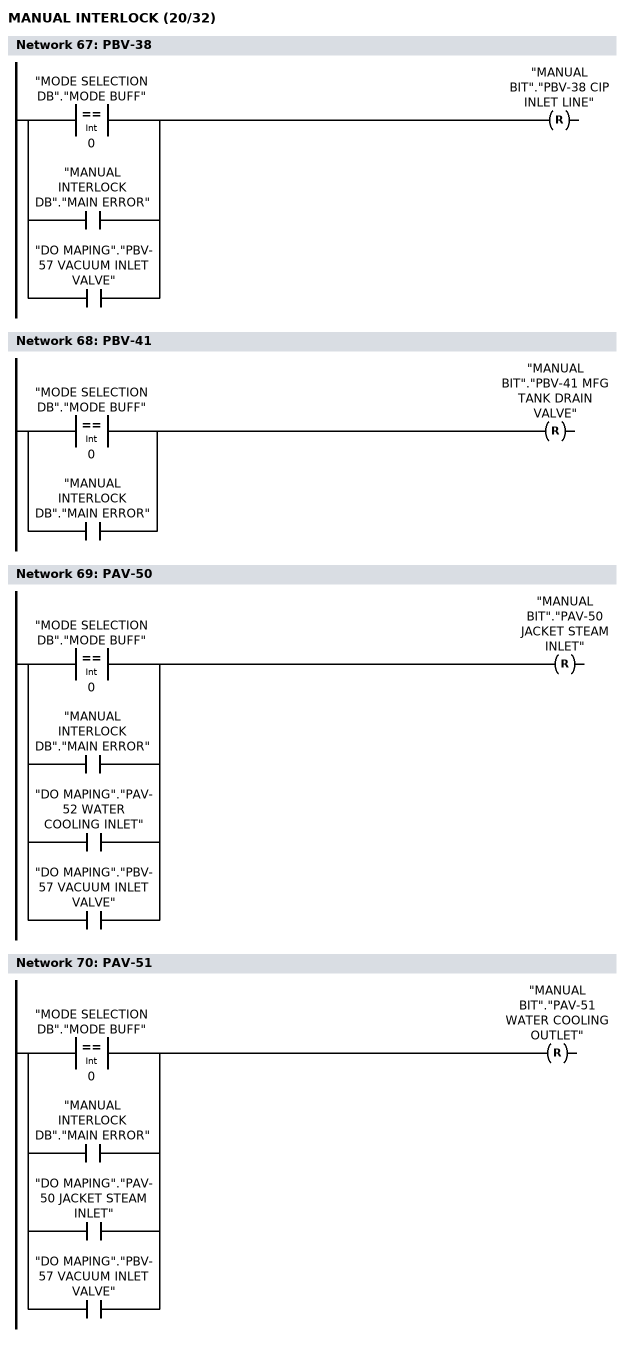
   RUNG wire#powerrail
      { S7_Templates := "SrcType := Int" } EQ_Contact(in1 := "MODE SELECTION DB"."MODE BUFF", in2 := 0)
      wire#w1
      R_Coil( "MANUAL BIT"."PBV-38 CIP INLET LINE" )
   END_RUNG
   RUNG wire#powerrail
      Contact( "MANUAL INTERLOCK DB"."MAIN ERROR" )
   END_RUNG wire#w1
   RUNG wire#powerrail
      Contact( "DO MAPING"."PBV-57 VACUUM INLET VALVE" )
   END_RUNG wire#w1
   // the same network as SCL:
   IF ("MODE SELECTION DB"."MODE BUFF" = 0) OR "MANUAL INTERLOCK DB"."MAIN ERROR" OR "DO MAPING"."PBV-57 VACUUM INLET VALVE" THEN
       "MANUAL BIT"."PBV-38 CIP INLET LINE" := FALSE;
   END_IF;
END_REGION

REGION Network 68: PBV-41
   RUNG wire#powerrail
      { S7_Templates := "SrcType := Int" } EQ_Contact(in1 := "MODE SELECTION DB"."MODE BUFF", in2 := 0)
      wire#w1
      R_Coil( "MANUAL BIT"."PBV-41 MFG TANK DRAIN VALVE" )
   END_RUNG
   RUNG wire#powerrail
      Contact( "MANUAL INTERLOCK DB"."MAIN ERROR" )
   END_RUNG wire#w1
   // the same network as SCL:
   IF ("MODE SELECTION DB"."MODE BUFF" = 0) OR "MANUAL INTERLOCK DB"."MAIN ERROR" THEN
       "MANUAL BIT"."PBV-41 MFG TANK DRAIN VALVE" := FALSE;
   END_IF;
END_REGION

REGION Network 69: PAV-50
   RUNG wire#powerrail
      { S7_Templates := "SrcType := Int" } EQ_Contact(in1 := "MODE SELECTION DB"."MODE BUFF", in2 := 0)
      wire#w1
      R_Coil( "MANUAL BIT"."PAV-50 JACKET STEAM INLET" )
   END_RUNG
   RUNG wire#powerrail
      Contact( "MANUAL INTERLOCK DB"."MAIN ERROR" )
   END_RUNG wire#w1
   RUNG wire#powerrail
      Contact( "DO MAPING"."PAV-52 WATER COOLING INLET" )
   END_RUNG wire#w1
   RUNG wire#powerrail
      Contact( "DO MAPING"."PBV-57 VACUUM INLET VALVE" )
   END_RUNG wire#w1
   // the same network as SCL:
   IF ("MODE SELECTION DB"."MODE BUFF" = 0) OR "MANUAL INTERLOCK DB"."MAIN ERROR" OR "DO MAPING"."PAV-52 WATER COOLING INLET" OR "DO MAPING"."PBV-57 VACUUM INLET VALVE" THEN
       "MANUAL BIT"."PAV-50 JACKET STEAM INLET" := FALSE;
   END_IF;
END_REGION

REGION Network 70: PAV-51
   RUNG wire#powerrail
      { S7_Templates := "SrcType := Int" } EQ_Contact(in1 := "MODE SELECTION DB"."MODE BUFF", in2 := 0)
      wire#w1
      R_Coil( "MANUAL BIT"."PAV-51 WATER COOLING OUTLET" )
   END_RUNG
   RUNG wire#powerrail
      Contact( "MANUAL INTERLOCK DB"."MAIN ERROR" )
   END_RUNG wire#w1
   RUNG wire#powerrail
      Contact( "DO MAPING"."PAV-50 JACKET STEAM INLET" )
   END_RUNG wire#w1
   RUNG wire#powerrail
      Contact( "DO MAPING"."PBV-57 VACUUM INLET VALVE" )
   END_RUNG wire#w1
   // the same network as SCL:
   IF ("MODE SELECTION DB"."MODE BUFF" = 0) OR "MANUAL INTERLOCK DB"."MAIN ERROR" OR "DO MAPING"."PAV-50 JACKET STEAM INLET" OR "DO MAPING"."PBV-57 VACUUM INLET VALVE" THEN
       "MANUAL BIT"."PAV-51 WATER COOLING OUTLET" := FALSE;
   END_IF;
END_REGION

REGION Network 71: PAV-52
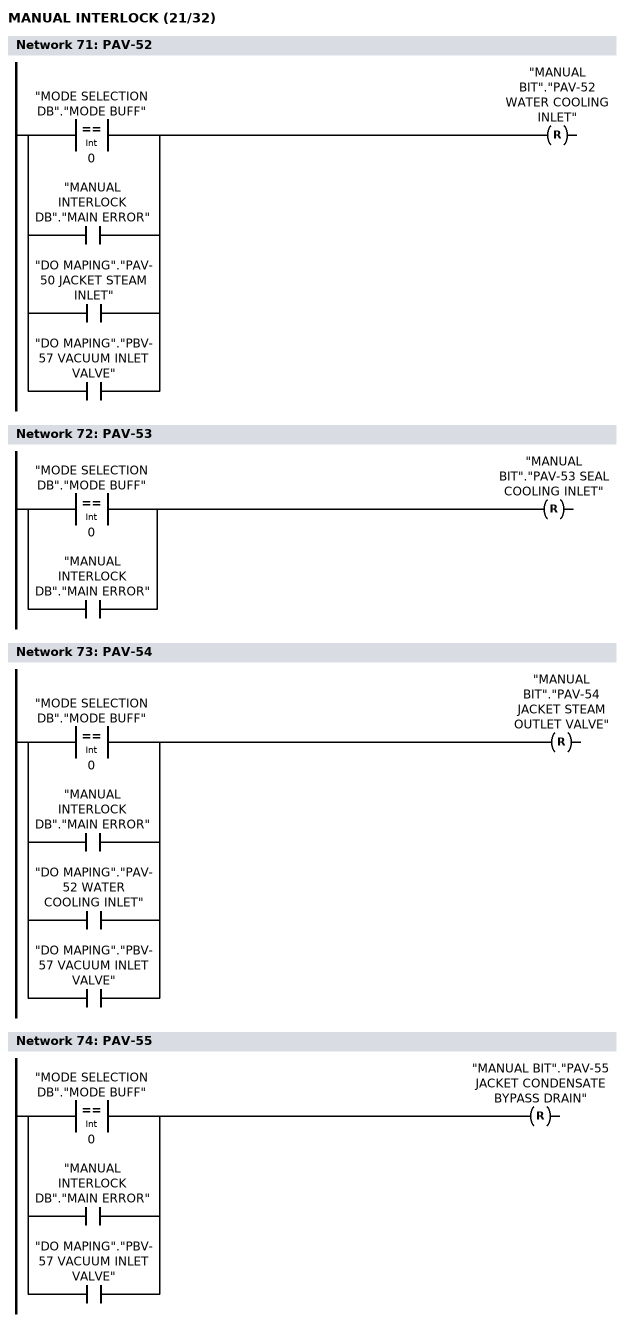
   RUNG wire#powerrail
      { S7_Templates := "SrcType := Int" } EQ_Contact(in1 := "MODE SELECTION DB"."MODE BUFF", in2 := 0)
      wire#w1
      R_Coil( "MANUAL BIT"."PAV-52 WATER COOLING INLET" )
   END_RUNG
   RUNG wire#powerrail
      Contact( "MANUAL INTERLOCK DB"."MAIN ERROR" )
   END_RUNG wire#w1
   RUNG wire#powerrail
      Contact( "DO MAPING"."PAV-50 JACKET STEAM INLET" )
   END_RUNG wire#w1
   RUNG wire#powerrail
      Contact( "DO MAPING"."PBV-57 VACUUM INLET VALVE" )
   END_RUNG wire#w1
   // the same network as SCL:
   IF ("MODE SELECTION DB"."MODE BUFF" = 0) OR "MANUAL INTERLOCK DB"."MAIN ERROR" OR "DO MAPING"."PAV-50 JACKET STEAM INLET" OR "DO MAPING"."PBV-57 VACUUM INLET VALVE" THEN
       "MANUAL BIT"."PAV-52 WATER COOLING INLET" := FALSE;
   END_IF;
END_REGION

REGION Network 72: PAV-53
   RUNG wire#powerrail
      { S7_Templates := "SrcType := Int" } EQ_Contact(in1 := "MODE SELECTION DB"."MODE BUFF", in2 := 0)
      wire#w1
      R_Coil( "MANUAL BIT"."PAV-53 SEAL COOLING INLET" )
   END_RUNG
   RUNG wire#powerrail
      Contact( "MANUAL INTERLOCK DB"."MAIN ERROR" )
   END_RUNG wire#w1
   // the same network as SCL:
   IF ("MODE SELECTION DB"."MODE BUFF" = 0) OR "MANUAL INTERLOCK DB"."MAIN ERROR" THEN
       "MANUAL BIT"."PAV-53 SEAL COOLING INLET" := FALSE;
   END_IF;
END_REGION

REGION Network 73: PAV-54
   RUNG wire#powerrail
      { S7_Templates := "SrcType := Int" } EQ_Contact(in1 := "MODE SELECTION DB"."MODE BUFF", in2 := 0)
      wire#w1
      R_Coil( "MANUAL BIT"."PAV-54 JACKET STEAM OUTLET VALVE" )
   END_RUNG
   RUNG wire#powerrail
      Contact( "MANUAL INTERLOCK DB"."MAIN ERROR" )
   END_RUNG wire#w1
   RUNG wire#powerrail
      Contact( "DO MAPING"."PAV-52 WATER COOLING INLET" )
   END_RUNG wire#w1
   RUNG wire#powerrail
      Contact( "DO MAPING"."PBV-57 VACUUM INLET VALVE" )
   END_RUNG wire#w1
   // the same network as SCL:
   IF ("MODE SELECTION DB"."MODE BUFF" = 0) OR "MANUAL INTERLOCK DB"."MAIN ERROR" OR "DO MAPING"."PAV-52 WATER COOLING INLET" OR "DO MAPING"."PBV-57 VACUUM INLET VALVE" THEN
       "MANUAL BIT"."PAV-54 JACKET STEAM OUTLET VALVE" := FALSE;
   END_IF;
END_REGION

REGION Network 74: PAV-55
   RUNG wire#powerrail
      { S7_Templates := "SrcType := Int" } EQ_Contact(in1 := "MODE SELECTION DB"."MODE BUFF", in2 := 0)
      wire#w1
      R_Coil( "MANUAL BIT"."PAV-55 JACKET CONDENSATE BYPASS DRAIN" )
   END_RUNG
   RUNG wire#powerrail
      Contact( "MANUAL INTERLOCK DB"."MAIN ERROR" )
   END_RUNG wire#w1
   RUNG wire#powerrail
      Contact( "DO MAPING"."PBV-57 VACUUM INLET VALVE" )
   END_RUNG wire#w1
   // the same network as SCL:
   IF ("MODE SELECTION DB"."MODE BUFF" = 0) OR "MANUAL INTERLOCK DB"."MAIN ERROR" OR "DO MAPING"."PBV-57 VACUUM INLET VALVE" THEN
       "MANUAL BIT"."PAV-55 JACKET CONDENSATE BYPASS DRAIN" := FALSE;
   END_IF;
END_REGION

REGION Network 75: PAV-56
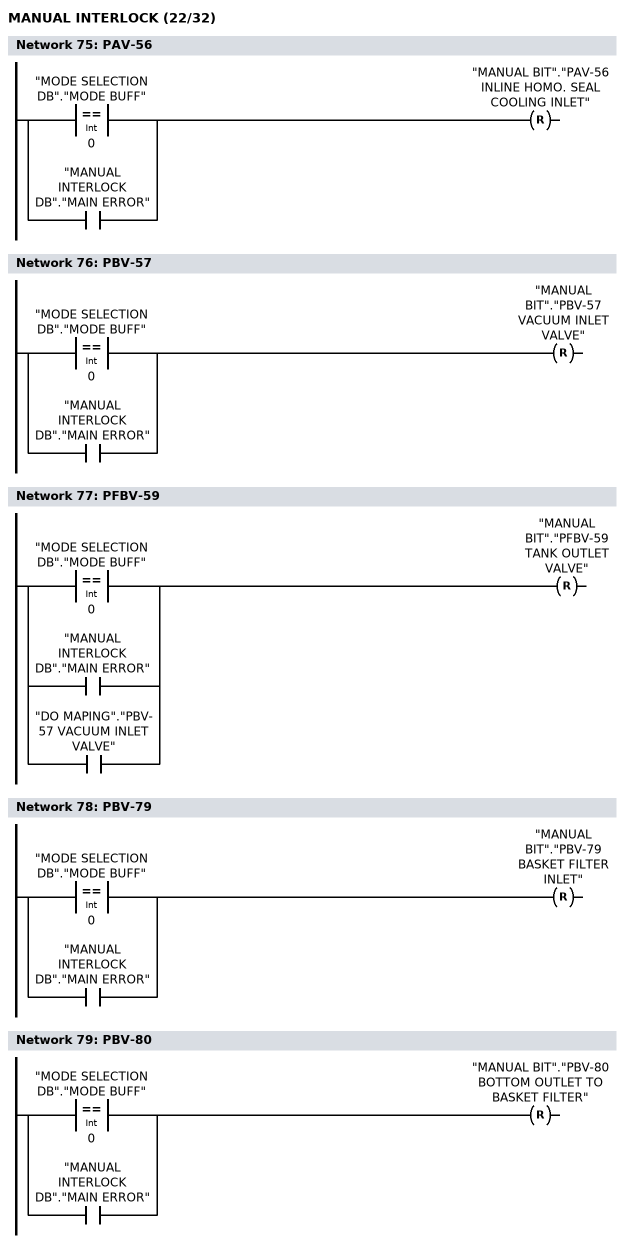
   RUNG wire#powerrail
      { S7_Templates := "SrcType := Int" } EQ_Contact(in1 := "MODE SELECTION DB"."MODE BUFF", in2 := 0)
      wire#w1
      R_Coil( "MANUAL BIT"."PAV-56 INLINE HOMO. SEAL COOLING INLET" )
   END_RUNG
   RUNG wire#powerrail
      Contact( "MANUAL INTERLOCK DB"."MAIN ERROR" )
   END_RUNG wire#w1
   // the same network as SCL:
   IF ("MODE SELECTION DB"."MODE BUFF" = 0) OR "MANUAL INTERLOCK DB"."MAIN ERROR" THEN
       "MANUAL BIT"."PAV-56 INLINE HOMO. SEAL COOLING INLET" := FALSE;
   END_IF;
END_REGION

REGION Network 76: PBV-57
   RUNG wire#powerrail
      { S7_Templates := "SrcType := Int" } EQ_Contact(in1 := "MODE SELECTION DB"."MODE BUFF", in2 := 0)
      wire#w1
      R_Coil( "MANUAL BIT"."PBV-57 VACUUM INLET VALVE" )
   END_RUNG
   RUNG wire#powerrail
      Contact( "MANUAL INTERLOCK DB"."MAIN ERROR" )
   END_RUNG wire#w1
   // the same network as SCL:
   IF ("MODE SELECTION DB"."MODE BUFF" = 0) OR "MANUAL INTERLOCK DB"."MAIN ERROR" THEN
       "MANUAL BIT"."PBV-57 VACUUM INLET VALVE" := FALSE;
   END_IF;
END_REGION

REGION Network 77: PFBV-59
   RUNG wire#powerrail
      { S7_Templates := "SrcType := Int" } EQ_Contact(in1 := "MODE SELECTION DB"."MODE BUFF", in2 := 0)
      wire#w1
      R_Coil( "MANUAL BIT"."PFBV-59 TANK OUTLET VALVE" )
   END_RUNG
   RUNG wire#powerrail
      Contact( "MANUAL INTERLOCK DB"."MAIN ERROR" )
   END_RUNG wire#w1
   RUNG wire#powerrail
      Contact( "DO MAPING"."PBV-57 VACUUM INLET VALVE" )
   END_RUNG wire#w1
   // the same network as SCL:
   IF ("MODE SELECTION DB"."MODE BUFF" = 0) OR "MANUAL INTERLOCK DB"."MAIN ERROR" OR "DO MAPING"."PBV-57 VACUUM INLET VALVE" THEN
       "MANUAL BIT"."PFBV-59 TANK OUTLET VALVE" := FALSE;
   END_IF;
END_REGION

REGION Network 78: PBV-79
   RUNG wire#powerrail
      { S7_Templates := "SrcType := Int" } EQ_Contact(in1 := "MODE SELECTION DB"."MODE BUFF", in2 := 0)
      wire#w1
      R_Coil( "MANUAL BIT"."PBV-79 BASKET FILTER INLET" )
   END_RUNG
   RUNG wire#powerrail
      Contact( "MANUAL INTERLOCK DB"."MAIN ERROR" )
   END_RUNG wire#w1
   // the same network as SCL:
   IF ("MODE SELECTION DB"."MODE BUFF" = 0) OR "MANUAL INTERLOCK DB"."MAIN ERROR" THEN
       "MANUAL BIT"."PBV-79 BASKET FILTER INLET" := FALSE;
   END_IF;
END_REGION

REGION Network 79: PBV-80
   RUNG wire#powerrail
      { S7_Templates := "SrcType := Int" } EQ_Contact(in1 := "MODE SELECTION DB"."MODE BUFF", in2 := 0)
      wire#w1
      R_Coil( "MANUAL BIT"."PBV-80 BOTTOM OUTLET TO BASKET FILTER" )
   END_RUNG
   RUNG wire#powerrail
      Contact( "MANUAL INTERLOCK DB"."MAIN ERROR" )
   END_RUNG wire#w1
   // the same network as SCL:
   IF ("MODE SELECTION DB"."MODE BUFF" = 0) OR "MANUAL INTERLOCK DB"."MAIN ERROR" THEN
       "MANUAL BIT"."PBV-80 BOTTOM OUTLET TO BASKET FILTER" := FALSE;
   END_IF;
END_REGION

REGION Network 80: PBV-81
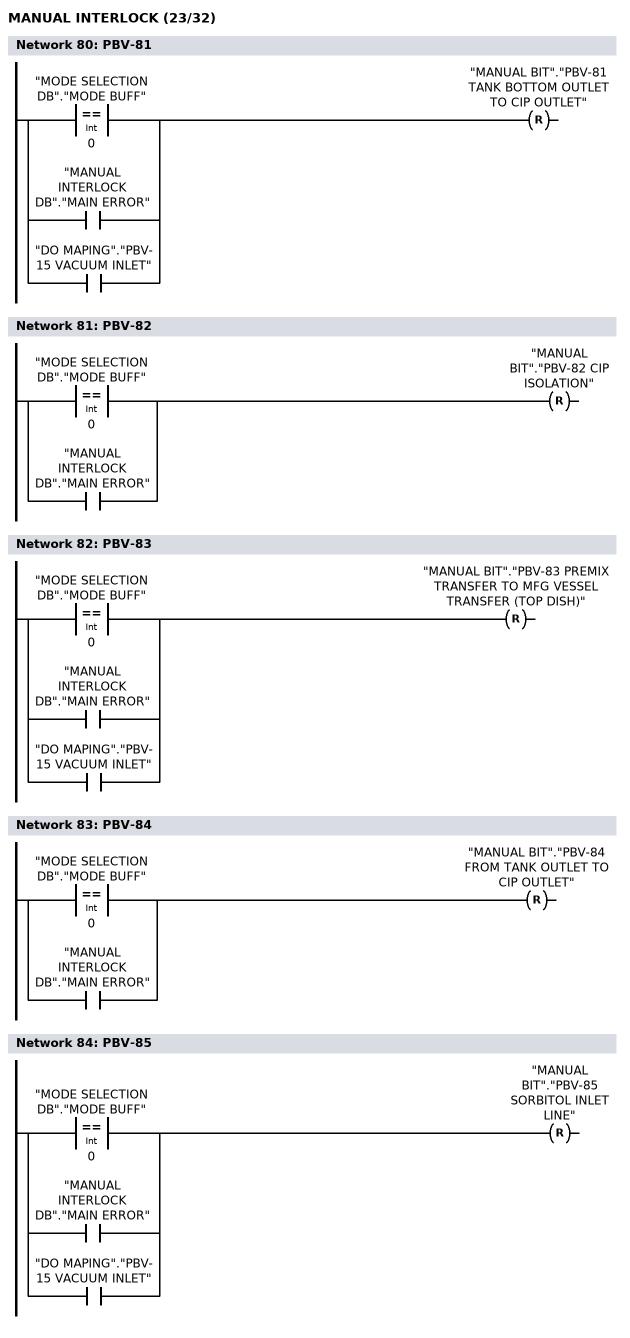
   RUNG wire#powerrail
      { S7_Templates := "SrcType := Int" } EQ_Contact(in1 := "MODE SELECTION DB"."MODE BUFF", in2 := 0)
      wire#w1
      R_Coil( "MANUAL BIT"."PBV-81 TANK BOTTOM OUTLET TO CIP OUTLET" )
   END_RUNG
   RUNG wire#powerrail
      Contact( "MANUAL INTERLOCK DB"."MAIN ERROR" )
   END_RUNG wire#w1
   RUNG wire#powerrail
      Contact( "DO MAPING"."PBV-15 VACUUM INLET" )
   END_RUNG wire#w1
   // the same network as SCL:
   IF ("MODE SELECTION DB"."MODE BUFF" = 0) OR "MANUAL INTERLOCK DB"."MAIN ERROR" OR "DO MAPING"."PBV-15 VACUUM INLET" THEN
       "MANUAL BIT"."PBV-81 TANK BOTTOM OUTLET TO CIP OUTLET" := FALSE;
   END_IF;
END_REGION

REGION Network 81: PBV-82
   RUNG wire#powerrail
      { S7_Templates := "SrcType := Int" } EQ_Contact(in1 := "MODE SELECTION DB"."MODE BUFF", in2 := 0)
      wire#w1
      R_Coil( "MANUAL BIT"."PBV-82 CIP ISOLATION" )
   END_RUNG
   RUNG wire#powerrail
      Contact( "MANUAL INTERLOCK DB"."MAIN ERROR" )
   END_RUNG wire#w1
   // the same network as SCL:
   IF ("MODE SELECTION DB"."MODE BUFF" = 0) OR "MANUAL INTERLOCK DB"."MAIN ERROR" THEN
       "MANUAL BIT"."PBV-82 CIP ISOLATION" := FALSE;
   END_IF;
END_REGION

REGION Network 82: PBV-83
   RUNG wire#powerrail
      { S7_Templates := "SrcType := Int" } EQ_Contact(in1 := "MODE SELECTION DB"."MODE BUFF", in2 := 0)
      wire#w1
      R_Coil( "MANUAL BIT"."PBV-83 PREMIX TRANSFER TO MFG VESSEL TRANSFER (TOP DISH)" )
   END_RUNG
   RUNG wire#powerrail
      Contact( "MANUAL INTERLOCK DB"."MAIN ERROR" )
   END_RUNG wire#w1
   RUNG wire#powerrail
      Contact( "DO MAPING"."PBV-15 VACUUM INLET" )
   END_RUNG wire#w1
   // the same network as SCL:
   IF ("MODE SELECTION DB"."MODE BUFF" = 0) OR "MANUAL INTERLOCK DB"."MAIN ERROR" OR "DO MAPING"."PBV-15 VACUUM INLET" THEN
       "MANUAL BIT"."PBV-83 PREMIX TRANSFER TO MFG VESSEL TRANSFER (TOP DISH)" := FALSE;
   END_IF;
END_REGION

REGION Network 83: PBV-84
   RUNG wire#powerrail
      { S7_Templates := "SrcType := Int" } EQ_Contact(in1 := "MODE SELECTION DB"."MODE BUFF", in2 := 0)
      wire#w1
      R_Coil( "MANUAL BIT"."PBV-84 FROM TANK OUTLET TO CIP OUTLET" )
   END_RUNG
   RUNG wire#powerrail
      Contact( "MANUAL INTERLOCK DB"."MAIN ERROR" )
   END_RUNG wire#w1
   // the same network as SCL:
   IF ("MODE SELECTION DB"."MODE BUFF" = 0) OR "MANUAL INTERLOCK DB"."MAIN ERROR" THEN
       "MANUAL BIT"."PBV-84 FROM TANK OUTLET TO CIP OUTLET" := FALSE;
   END_IF;
END_REGION

REGION Network 84: PBV-85
   RUNG wire#powerrail
      { S7_Templates := "SrcType := Int" } EQ_Contact(in1 := "MODE SELECTION DB"."MODE BUFF", in2 := 0)
      wire#w1
      R_Coil( "MANUAL BIT"."PBV-85 SORBITOL INLET LINE" )
   END_RUNG
   RUNG wire#powerrail
      Contact( "MANUAL INTERLOCK DB"."MAIN ERROR" )
   END_RUNG wire#w1
   RUNG wire#powerrail
      Contact( "DO MAPING"."PBV-15 VACUUM INLET" )
   END_RUNG wire#w1
   // the same network as SCL:
   IF ("MODE SELECTION DB"."MODE BUFF" = 0) OR "MANUAL INTERLOCK DB"."MAIN ERROR" OR "DO MAPING"."PBV-15 VACUUM INLET" THEN
       "MANUAL BIT"."PBV-85 SORBITOL INLET LINE" := FALSE;
   END_IF;
END_REGION

REGION Network 85: PBV-86
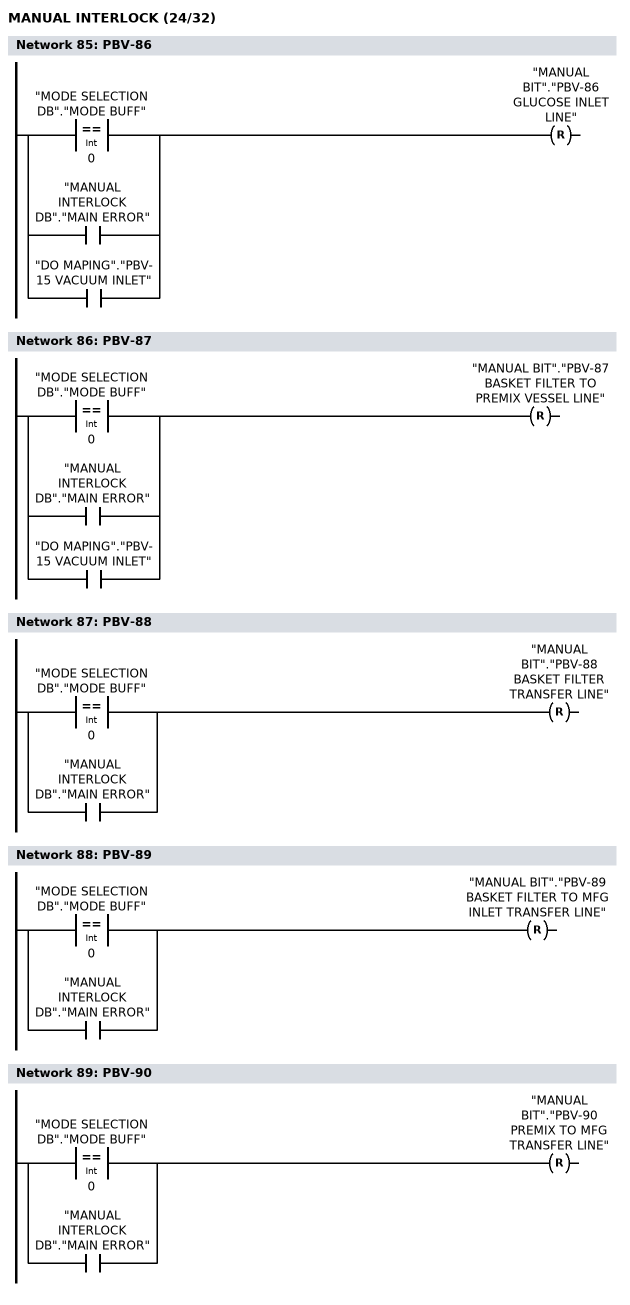
   RUNG wire#powerrail
      { S7_Templates := "SrcType := Int" } EQ_Contact(in1 := "MODE SELECTION DB"."MODE BUFF", in2 := 0)
      wire#w1
      R_Coil( "MANUAL BIT"."PBV-86 GLUCOSE INLET LINE" )
   END_RUNG
   RUNG wire#powerrail
      Contact( "MANUAL INTERLOCK DB"."MAIN ERROR" )
   END_RUNG wire#w1
   RUNG wire#powerrail
      Contact( "DO MAPING"."PBV-15 VACUUM INLET" )
   END_RUNG wire#w1
   // the same network as SCL:
   IF ("MODE SELECTION DB"."MODE BUFF" = 0) OR "MANUAL INTERLOCK DB"."MAIN ERROR" OR "DO MAPING"."PBV-15 VACUUM INLET" THEN
       "MANUAL BIT"."PBV-86 GLUCOSE INLET LINE" := FALSE;
   END_IF;
END_REGION

REGION Network 86: PBV-87
   RUNG wire#powerrail
      { S7_Templates := "SrcType := Int" } EQ_Contact(in1 := "MODE SELECTION DB"."MODE BUFF", in2 := 0)
      wire#w1
      R_Coil( "MANUAL BIT"."PBV-87 BASKET FILTER TO PREMIX VESSEL LINE" )
   END_RUNG
   RUNG wire#powerrail
      Contact( "MANUAL INTERLOCK DB"."MAIN ERROR" )
   END_RUNG wire#w1
   RUNG wire#powerrail
      Contact( "DO MAPING"."PBV-15 VACUUM INLET" )
   END_RUNG wire#w1
   // the same network as SCL:
   IF ("MODE SELECTION DB"."MODE BUFF" = 0) OR "MANUAL INTERLOCK DB"."MAIN ERROR" OR "DO MAPING"."PBV-15 VACUUM INLET" THEN
       "MANUAL BIT"."PBV-87 BASKET FILTER TO PREMIX VESSEL LINE" := FALSE;
   END_IF;
END_REGION

REGION Network 87: PBV-88
   RUNG wire#powerrail
      { S7_Templates := "SrcType := Int" } EQ_Contact(in1 := "MODE SELECTION DB"."MODE BUFF", in2 := 0)
      wire#w1
      R_Coil( "MANUAL BIT"."PBV-88 BASKET FILTER TRANSFER LINE" )
   END_RUNG
   RUNG wire#powerrail
      Contact( "MANUAL INTERLOCK DB"."MAIN ERROR" )
   END_RUNG wire#w1
   // the same network as SCL:
   IF ("MODE SELECTION DB"."MODE BUFF" = 0) OR "MANUAL INTERLOCK DB"."MAIN ERROR" THEN
       "MANUAL BIT"."PBV-88 BASKET FILTER TRANSFER LINE" := FALSE;
   END_IF;
END_REGION

REGION Network 88: PBV-89
   RUNG wire#powerrail
      { S7_Templates := "SrcType := Int" } EQ_Contact(in1 := "MODE SELECTION DB"."MODE BUFF", in2 := 0)
      wire#w1
      R_Coil( "MANUAL BIT"."PBV-89 BASKET FILTER TO MFG INLET TRANSFER LINE" )
   END_RUNG
   RUNG wire#powerrail
      Contact( "MANUAL INTERLOCK DB"."MAIN ERROR" )
   END_RUNG wire#w1
   // the same network as SCL:
   IF ("MODE SELECTION DB"."MODE BUFF" = 0) OR "MANUAL INTERLOCK DB"."MAIN ERROR" THEN
       "MANUAL BIT"."PBV-89 BASKET FILTER TO MFG INLET TRANSFER LINE" := FALSE;
   END_IF;
END_REGION

REGION Network 89: PBV-90
   RUNG wire#powerrail
      { S7_Templates := "SrcType := Int" } EQ_Contact(in1 := "MODE SELECTION DB"."MODE BUFF", in2 := 0)
      wire#w1
      R_Coil( "MANUAL BIT"."PBV-90 PREMIX TO MFG TRANSFER LINE" )
   END_RUNG
   RUNG wire#powerrail
      Contact( "MANUAL INTERLOCK DB"."MAIN ERROR" )
   END_RUNG wire#w1
   // the same network as SCL:
   IF ("MODE SELECTION DB"."MODE BUFF" = 0) OR "MANUAL INTERLOCK DB"."MAIN ERROR" THEN
       "MANUAL BIT"."PBV-90 PREMIX TO MFG TRANSFER LINE" := FALSE;
   END_IF;
END_REGION

REGION Network 90: PBV-91
